METHOD PUBLIC Check_LWORD_TO_BOOL_Max
VAR
	value : LWORD := DatatypeLimits.LWORD_MAX_VALUE;
	actual : BOOL;
	converted : BOOL;
	equal : BOOL;
END_VAR
TEST('Check_LWORD_TO_BOOL_Max');

// @TEST-RUN
converted := TryConvert_LWORD_TO_Destination(value, actual);
equal := actual = LWORD_TO_BOOL(value);

// @TEST-ASSERT
AssertTrue(Condition := equal, Message := 'Did not convert LWORD to BOOL correctly');
AssertTrue(Condition := converted, Message := 'Did not report LWORD to BOOL conversion was successful');

TEST_FINISHED();
END_METHOD

METHOD PUBLIC Check_LWORD_TO_BYTE_Min
VAR
	value : LWORD := DatatypeLimits.LWORD_MIN_VALUE;
	actual : BYTE;
	converted : BOOL;
	equal : BOOL;
END_VAR
TEST('Check_LWORD_TO_BYTE_Min');

// @TEST-RUN
converted := TryConvert_LWORD_TO_Destination(value, actual);
equal := actual = LWORD_TO_BYTE(value);

// @TEST-ASSERT
AssertTrue(Condition := equal, Message := 'Did not convert LWORD to BYTE correctly');
AssertTrue(Condition := converted, Message := 'Did not report LWORD to BYTE conversion was successful');

TEST_FINISHED();
END_METHOD

METHOD PUBLIC Check_LWORD_TO_BYTE_TooHigh
VAR
	value : LWORD := DatatypeLimits.LWORD_MAX_VALUE;
	actual : BYTE;
	converted : BOOL;
END_VAR
TEST('Check_LWORD_TO_BYTE_TooHigh');

// @TEST-RUN
converted := TryConvert_LWORD_TO_Destination(value, actual);

// @TEST-ASSERT
AssertFalse(Condition := converted, Message := 'Did not report LWORD to BYTE conversion was prevented');

TEST_FINISHED();
END_METHOD

METHOD PUBLIC Check_LWORD_TO_BYTE_Max
VAR
	value : LWORD := DatatypeLimits.MAX_VALUE_OF_LWORD_WHICH_CAN_BE_HELD_IN_A_BYTE;
	actual : BYTE;
	converted : BOOL;
	equal : BOOL;
END_VAR
TEST('Check_LWORD_TO_BYTE_Max');

// @TEST-RUN
converted := TryConvert_LWORD_TO_Destination(value, actual);
equal := actual = LWORD_TO_BYTE(value);

// @TEST-ASSERT
AssertTrue(Condition := equal, Message := 'Did not convert LWORD to BYTE correctly');
AssertTrue(Condition := converted, Message := 'Did not report LWORD to BYTE conversion was successful');

TEST_FINISHED();
END_METHOD

METHOD PUBLIC Check_LWORD_TO_DATE_Min
VAR
	value : LWORD := DatatypeLimits.LWORD_MIN_VALUE;
	actual : DATE;
	converted : BOOL;
	equal : BOOL;
END_VAR
TEST('Check_LWORD_TO_DATE_Min');

// @TEST-RUN
converted := TryConvert_LWORD_TO_Destination(value, actual);
equal := actual = LWORD_TO_DATE(value);

// @TEST-ASSERT
AssertTrue(Condition := equal, Message := 'Did not convert LWORD to DATE correctly');
AssertTrue(Condition := converted, Message := 'Did not report LWORD to DATE conversion was successful');

TEST_FINISHED();
END_METHOD

METHOD PUBLIC Check_LWORD_TO_DATE_TooHigh
VAR
	value : LWORD := DatatypeLimits.LWORD_MAX_VALUE;
	actual : DATE;
	converted : BOOL;
END_VAR
TEST('Check_LWORD_TO_DATE_TooHigh');

// @TEST-RUN
converted := TryConvert_LWORD_TO_Destination(value, actual);

// @TEST-ASSERT
AssertFalse(Condition := converted, Message := 'Did not report LWORD to DATE conversion was prevented');

TEST_FINISHED();
END_METHOD

METHOD PUBLIC Check_LWORD_TO_DATE_Max
VAR
	value : LWORD := DatatypeLimits.MAX_VALUE_OF_LWORD_WHICH_CAN_BE_HELD_IN_A_DATE;
	actual : DATE;
	converted : BOOL;
	equal : BOOL;
END_VAR
TEST('Check_LWORD_TO_DATE_Max');

// @TEST-RUN
converted := TryConvert_LWORD_TO_Destination(value, actual);
equal := actual = LWORD_TO_DATE(value);

// @TEST-ASSERT
AssertTrue(Condition := equal, Message := 'Did not convert LWORD to DATE correctly');
AssertTrue(Condition := converted, Message := 'Did not report LWORD to DATE conversion was successful');

TEST_FINISHED();
END_METHOD

METHOD PUBLIC Check_LWORD_TO_DINT_Min
VAR
	value : LWORD := DatatypeLimits.LWORD_MIN_VALUE;
	actual : DINT;
	converted : BOOL;
	equal : BOOL;
END_VAR
TEST('Check_LWORD_TO_DINT_Min');

// @TEST-RUN
converted := TryConvert_LWORD_TO_Destination(value, actual);
equal := actual = LWORD_TO_DINT(value);

// @TEST-ASSERT
AssertTrue(Condition := equal, Message := 'Did not convert LWORD to DINT correctly');
AssertTrue(Condition := converted, Message := 'Did not report LWORD to DINT conversion was successful');

TEST_FINISHED();
END_METHOD

METHOD PUBLIC Check_LWORD_TO_DINT_TooHigh
VAR
	value : LWORD := DatatypeLimits.LWORD_MAX_VALUE;
	actual : DINT;
	converted : BOOL;
END_VAR
TEST('Check_LWORD_TO_DINT_TooHigh');

// @TEST-RUN
converted := TryConvert_LWORD_TO_Destination(value, actual);

// @TEST-ASSERT
AssertFalse(Condition := converted, Message := 'Did not report LWORD to DINT conversion was prevented');

TEST_FINISHED();
END_METHOD

METHOD PUBLIC Check_LWORD_TO_DINT_Max
VAR
	value : LWORD := DatatypeLimits.MAX_VALUE_OF_LWORD_WHICH_CAN_BE_HELD_IN_A_DINT;
	actual : DINT;
	converted : BOOL;
	equal : BOOL;
END_VAR
TEST('Check_LWORD_TO_DINT_Max');

// @TEST-RUN
converted := TryConvert_LWORD_TO_Destination(value, actual);
equal := actual = LWORD_TO_DINT(value);

// @TEST-ASSERT
AssertTrue(Condition := equal, Message := 'Did not convert LWORD to DINT correctly');
AssertTrue(Condition := converted, Message := 'Did not report LWORD to DINT conversion was successful');

TEST_FINISHED();
END_METHOD

METHOD PUBLIC Check_LWORD_TO_DT_Min
VAR
	value : LWORD := DatatypeLimits.LWORD_MIN_VALUE;
	actual : DT;
	converted : BOOL;
	equal : BOOL;
END_VAR
TEST('Check_LWORD_TO_DT_Min');

// @TEST-RUN
converted := TryConvert_LWORD_TO_Destination(value, actual);
equal := actual = LWORD_TO_DT(value);

// @TEST-ASSERT
AssertTrue(Condition := equal, Message := 'Did not convert LWORD to DT correctly');
AssertTrue(Condition := converted, Message := 'Did not report LWORD to DT conversion was successful');

TEST_FINISHED();
END_METHOD

METHOD PUBLIC Check_LWORD_TO_DT_TooHigh
VAR
	value : LWORD := DatatypeLimits.LWORD_MAX_VALUE;
	actual : DT;
	converted : BOOL;
END_VAR
TEST('Check_LWORD_TO_DT_TooHigh');

// @TEST-RUN
converted := TryConvert_LWORD_TO_Destination(value, actual);

// @TEST-ASSERT
AssertFalse(Condition := converted, Message := 'Did not report LWORD to DT conversion was prevented');

TEST_FINISHED();
END_METHOD

METHOD PUBLIC Check_LWORD_TO_DT_Max
VAR
	value : LWORD := DatatypeLimits.MAX_VALUE_OF_LWORD_WHICH_CAN_BE_HELD_IN_A_DT;
	actual : DT;
	converted : BOOL;
	equal : BOOL;
END_VAR
TEST('Check_LWORD_TO_DT_Max');

// @TEST-RUN
converted := TryConvert_LWORD_TO_Destination(value, actual);
equal := actual = LWORD_TO_DT(value);

// @TEST-ASSERT
AssertTrue(Condition := equal, Message := 'Did not convert LWORD to DT correctly');
AssertTrue(Condition := converted, Message := 'Did not report LWORD to DT conversion was successful');

TEST_FINISHED();
END_METHOD

METHOD PUBLIC Check_LWORD_TO_DWORD_Min
VAR
	value : LWORD := DatatypeLimits.LWORD_MIN_VALUE;
	actual : DWORD;
	converted : BOOL;
	equal : BOOL;
END_VAR
TEST('Check_LWORD_TO_DWORD_Min');

// @TEST-RUN
converted := TryConvert_LWORD_TO_Destination(value, actual);
equal := actual = LWORD_TO_DWORD(value);

// @TEST-ASSERT
AssertTrue(Condition := equal, Message := 'Did not convert LWORD to DWORD correctly');
AssertTrue(Condition := converted, Message := 'Did not report LWORD to DWORD conversion was successful');

TEST_FINISHED();
END_METHOD

METHOD PUBLIC Check_LWORD_TO_DWORD_TooHigh
VAR
	value : LWORD := DatatypeLimits.LWORD_MAX_VALUE;
	actual : DWORD;
	converted : BOOL;
END_VAR
TEST('Check_LWORD_TO_DWORD_TooHigh');

// @TEST-RUN
converted := TryConvert_LWORD_TO_Destination(value, actual);

// @TEST-ASSERT
AssertFalse(Condition := converted, Message := 'Did not report LWORD to DWORD conversion was prevented');

TEST_FINISHED();
END_METHOD

METHOD PUBLIC Check_LWORD_TO_DWORD_Max
VAR
	value : LWORD := DatatypeLimits.MAX_VALUE_OF_LWORD_WHICH_CAN_BE_HELD_IN_A_DWORD;
	actual : DWORD;
	converted : BOOL;
	equal : BOOL;
END_VAR
TEST('Check_LWORD_TO_DWORD_Max');

// @TEST-RUN
converted := TryConvert_LWORD_TO_Destination(value, actual);
equal := actual = LWORD_TO_DWORD(value);

// @TEST-ASSERT
AssertTrue(Condition := equal, Message := 'Did not convert LWORD to DWORD correctly');
AssertTrue(Condition := converted, Message := 'Did not report LWORD to DWORD conversion was successful');

TEST_FINISHED();
END_METHOD

METHOD PUBLIC Check_LWORD_TO_INT_Min
VAR
	value : LWORD := DatatypeLimits.LWORD_MIN_VALUE;
	actual : INT;
	converted : BOOL;
	equal : BOOL;
END_VAR
TEST('Check_LWORD_TO_INT_Min');

// @TEST-RUN
converted := TryConvert_LWORD_TO_Destination(value, actual);
equal := actual = LWORD_TO_INT(value);

// @TEST-ASSERT
AssertTrue(Condition := equal, Message := 'Did not convert LWORD to INT correctly');
AssertTrue(Condition := converted, Message := 'Did not report LWORD to INT conversion was successful');

TEST_FINISHED();
END_METHOD

METHOD PUBLIC Check_LWORD_TO_INT_TooHigh
VAR
	value : LWORD := DatatypeLimits.LWORD_MAX_VALUE;
	actual : INT;
	converted : BOOL;
END_VAR
TEST('Check_LWORD_TO_INT_TooHigh');

// @TEST-RUN
converted := TryConvert_LWORD_TO_Destination(value, actual);

// @TEST-ASSERT
AssertFalse(Condition := converted, Message := 'Did not report LWORD to INT conversion was prevented');

TEST_FINISHED();
END_METHOD

METHOD PUBLIC Check_LWORD_TO_INT_Max
VAR
	value : LWORD := DatatypeLimits.MAX_VALUE_OF_LWORD_WHICH_CAN_BE_HELD_IN_A_INT;
	actual : INT;
	converted : BOOL;
	equal : BOOL;
END_VAR
TEST('Check_LWORD_TO_INT_Max');

// @TEST-RUN
converted := TryConvert_LWORD_TO_Destination(value, actual);
equal := actual = LWORD_TO_INT(value);

// @TEST-ASSERT
AssertTrue(Condition := equal, Message := 'Did not convert LWORD to INT correctly');
AssertTrue(Condition := converted, Message := 'Did not report LWORD to INT conversion was successful');

TEST_FINISHED();
END_METHOD

METHOD PUBLIC Check_LWORD_TO_LINT_Min
VAR
	value : LWORD := DatatypeLimits.LWORD_MIN_VALUE;
	actual : LINT;
	converted : BOOL;
	equal : BOOL;
END_VAR
TEST('Check_LWORD_TO_LINT_Min');

// @TEST-RUN
converted := TryConvert_LWORD_TO_Destination(value, actual);
equal := actual = LWORD_TO_LINT(value);

// @TEST-ASSERT
AssertTrue(Condition := equal, Message := 'Did not convert LWORD to LINT correctly');
AssertTrue(Condition := converted, Message := 'Did not report LWORD to LINT conversion was successful');

TEST_FINISHED();
END_METHOD

METHOD PUBLIC Check_LWORD_TO_LINT_TooHigh
VAR
	value : LWORD := DatatypeLimits.LWORD_MAX_VALUE;
	actual : LINT;
	converted : BOOL;
END_VAR
TEST('Check_LWORD_TO_LINT_TooHigh');

// @TEST-RUN
converted := TryConvert_LWORD_TO_Destination(value, actual);

// @TEST-ASSERT
AssertFalse(Condition := converted, Message := 'Did not report LWORD to LINT conversion was prevented');

TEST_FINISHED();
END_METHOD

METHOD PUBLIC Check_LWORD_TO_LINT_Max
VAR
	value : LWORD := DatatypeLimits.MAX_VALUE_OF_LWORD_WHICH_CAN_BE_HELD_IN_A_LINT;
	actual : LINT;
	converted : BOOL;
	equal : BOOL;
END_VAR
TEST('Check_LWORD_TO_LINT_Max');

// @TEST-RUN
converted := TryConvert_LWORD_TO_Destination(value, actual);
equal := actual = LWORD_TO_LINT(value);

// @TEST-ASSERT
AssertTrue(Condition := equal, Message := 'Did not convert LWORD to LINT correctly');
AssertTrue(Condition := converted, Message := 'Did not report LWORD to LINT conversion was successful');

TEST_FINISHED();
END_METHOD

METHOD PUBLIC Check_LWORD_TO_LREAL_Min
VAR
	value : LWORD := DatatypeLimits.LWORD_MIN_VALUE;
	actual : LREAL;
	converted : BOOL;
	equal : BOOL;
END_VAR
TEST('Check_LWORD_TO_LREAL_Min');

// @TEST-RUN
converted := TryConvert_LWORD_TO_Destination(value, actual);
equal := actual = LWORD_TO_LREAL(value);

// @TEST-ASSERT
AssertTrue(Condition := equal, Message := 'Did not convert LWORD to LREAL correctly');
AssertTrue(Condition := converted, Message := 'Did not report LWORD to LREAL conversion was successful');

TEST_FINISHED();
END_METHOD

METHOD PUBLIC Check_LWORD_TO_LREAL_Max
VAR
	value : LWORD := DatatypeLimits.LWORD_MAX_VALUE;
	actual : LREAL;
	converted : BOOL;
	equal : BOOL;
END_VAR
TEST('Check_LWORD_TO_LREAL_Max');

// @TEST-RUN
converted := TryConvert_LWORD_TO_Destination(value, actual);
equal := actual = LWORD_TO_LREAL(value);

// @TEST-ASSERT
AssertTrue(Condition := equal, Message := 'Did not convert LWORD to LREAL correctly');
AssertTrue(Condition := converted, Message := 'Did not report LWORD to LREAL conversion was successful');

TEST_FINISHED();
END_METHOD

METHOD PUBLIC Check_LWORD_TO_LWORD_Min
VAR
	value : LWORD := DatatypeLimits.LWORD_MIN_VALUE;
	actual : LWORD;
	converted : BOOL;
	equal : BOOL;
END_VAR
TEST('Check_LWORD_TO_LWORD_Min');

// @TEST-RUN
converted := TryConvert_LWORD_TO_Destination(value, actual);
equal := actual = value;

// @TEST-ASSERT
AssertTrue(Condition := equal, Message := 'Did not convert LWORD to LWORD correctly');
AssertTrue(Condition := converted, Message := 'Did not report LWORD to LWORD conversion was successful');

TEST_FINISHED();
END_METHOD

METHOD PUBLIC Check_LWORD_TO_LWORD_Max
VAR
	value : LWORD := DatatypeLimits.LWORD_MAX_VALUE;
	actual : LWORD;
	converted : BOOL;
	equal : BOOL;
END_VAR
TEST('Check_LWORD_TO_LWORD_Max');

// @TEST-RUN
converted := TryConvert_LWORD_TO_Destination(value, actual);
equal := actual = value;

// @TEST-ASSERT
AssertTrue(Condition := equal, Message := 'Did not convert LWORD to LWORD correctly');
AssertTrue(Condition := converted, Message := 'Did not report LWORD to LWORD conversion was successful');

TEST_FINISHED();
END_METHOD

METHOD PUBLIC Check_LWORD_TO_REAL_Min
VAR
	value : LWORD := DatatypeLimits.LWORD_MIN_VALUE;
	actual : REAL;
	converted : BOOL;
	equal : BOOL;
END_VAR
TEST('Check_LWORD_TO_REAL_Min');

// @TEST-RUN
converted := TryConvert_LWORD_TO_Destination(value, actual);
equal := actual = LWORD_TO_REAL(value);

// @TEST-ASSERT
AssertTrue(Condition := equal, Message := 'Did not convert LWORD to REAL correctly');
AssertTrue(Condition := converted, Message := 'Did not report LWORD to REAL conversion was successful');

TEST_FINISHED();
END_METHOD

METHOD PUBLIC Check_LWORD_TO_REAL_Max
VAR
	value : LWORD := DatatypeLimits.LWORD_MAX_VALUE;
	actual : REAL;
	converted : BOOL;
	equal : BOOL;
END_VAR
TEST('Check_LWORD_TO_REAL_Max');

// @TEST-RUN
converted := TryConvert_LWORD_TO_Destination(value, actual);
equal := actual = LWORD_TO_REAL(value);

// @TEST-ASSERT
AssertTrue(Condition := equal, Message := 'Did not convert LWORD to REAL correctly');
AssertTrue(Condition := converted, Message := 'Did not report LWORD to REAL conversion was successful');

TEST_FINISHED();
END_METHOD

METHOD PUBLIC Check_LWORD_TO_SINT_Min
VAR
	value : LWORD := DatatypeLimits.LWORD_MIN_VALUE;
	actual : SINT;
	converted : BOOL;
	equal : BOOL;
END_VAR
TEST('Check_LWORD_TO_SINT_Min');

// @TEST-RUN
converted := TryConvert_LWORD_TO_Destination(value, actual);
equal := actual = LWORD_TO_SINT(value);

// @TEST-ASSERT
AssertTrue(Condition := equal, Message := 'Did not convert LWORD to SINT correctly');
AssertTrue(Condition := converted, Message := 'Did not report LWORD to SINT conversion was successful');

TEST_FINISHED();
END_METHOD

METHOD PUBLIC Check_LWORD_TO_SINT_TooHigh
VAR
	value : LWORD := DatatypeLimits.LWORD_MAX_VALUE;
	actual : SINT;
	converted : BOOL;
END_VAR
TEST('Check_LWORD_TO_SINT_TooHigh');

// @TEST-RUN
converted := TryConvert_LWORD_TO_Destination(value, actual);

// @TEST-ASSERT
AssertFalse(Condition := converted, Message := 'Did not report LWORD to SINT conversion was prevented');

TEST_FINISHED();
END_METHOD

METHOD PUBLIC Check_LWORD_TO_SINT_Max
VAR
	value : LWORD := DatatypeLimits.MAX_VALUE_OF_LWORD_WHICH_CAN_BE_HELD_IN_A_SINT;
	actual : SINT;
	converted : BOOL;
	equal : BOOL;
END_VAR
TEST('Check_LWORD_TO_SINT_Max');

// @TEST-RUN
converted := TryConvert_LWORD_TO_Destination(value, actual);
equal := actual = LWORD_TO_SINT(value);

// @TEST-ASSERT
AssertTrue(Condition := equal, Message := 'Did not convert LWORD to SINT correctly');
AssertTrue(Condition := converted, Message := 'Did not report LWORD to SINT conversion was successful');

TEST_FINISHED();
END_METHOD

METHOD PUBLIC Check_LWORD_TO_STRING_Min
VAR
	value : LWORD := DatatypeLimits.LWORD_MIN_VALUE;
	actual : STRING;
	converted : BOOL;
	equal : BOOL;
END_VAR
TEST('Check_LWORD_TO_STRING_Min');

// @TEST-RUN
converted := TryConvert_LWORD_TO_Destination(value, actual);
equal := actual = LWORD_TO_STRING(value);

// @TEST-ASSERT
AssertTrue(Condition := equal, Message := 'Did not convert LWORD to STRING correctly');
AssertTrue(Condition := converted, Message := 'Did not report LWORD to STRING conversion was successful');

TEST_FINISHED();
END_METHOD

METHOD PUBLIC Check_LWORD_TO_STRING_Max
VAR
	value : LWORD := DatatypeLimits.LWORD_MAX_VALUE;
	actual : STRING;
	converted : BOOL;
	equal : BOOL;
END_VAR
TEST('Check_LWORD_TO_STRING_Max');

// @TEST-RUN
converted := TryConvert_LWORD_TO_Destination(value, actual);
equal := actual = LWORD_TO_STRING(value);

// @TEST-ASSERT
AssertTrue(Condition := equal, Message := 'Did not convert LWORD to STRING correctly');
AssertTrue(Condition := converted, Message := 'Did not report LWORD to STRING conversion was successful');

TEST_FINISHED();
END_METHOD

METHOD PUBLIC Check_LWORD_TO_TIME_Min
VAR
	value : LWORD := DatatypeLimits.LWORD_MIN_VALUE;
	actual : TIME;
	converted : BOOL;
	equal : BOOL;
END_VAR
TEST('Check_LWORD_TO_TIME_Min');

// @TEST-RUN
converted := TryConvert_LWORD_TO_Destination(value, actual);
equal := actual = LWORD_TO_TIME(value);

// @TEST-ASSERT
AssertTrue(Condition := equal, Message := 'Did not convert LWORD to TIME correctly');
AssertTrue(Condition := converted, Message := 'Did not report LWORD to TIME conversion was successful');

TEST_FINISHED();
END_METHOD

METHOD PUBLIC Check_LWORD_TO_TIME_TooHigh
VAR
	value : LWORD := DatatypeLimits.LWORD_MAX_VALUE;
	actual : TIME;
	converted : BOOL;
END_VAR
TEST('Check_LWORD_TO_TIME_TooHigh');

// @TEST-RUN
converted := TryConvert_LWORD_TO_Destination(value, actual);

// @TEST-ASSERT
AssertFalse(Condition := converted, Message := 'Did not report LWORD to TIME conversion was prevented');

TEST_FINISHED();
END_METHOD

METHOD PUBLIC Check_LWORD_TO_TIME_Max
VAR
	value : LWORD := DatatypeLimits.MAX_VALUE_OF_LWORD_WHICH_CAN_BE_HELD_IN_A_TIME;
	actual : TIME;
	converted : BOOL;
	equal : BOOL;
END_VAR
TEST('Check_LWORD_TO_TIME_Max');

// @TEST-RUN
converted := TryConvert_LWORD_TO_Destination(value, actual);
equal := actual = LWORD_TO_TIME(value);

// @TEST-ASSERT
AssertTrue(Condition := equal, Message := 'Did not convert LWORD to TIME correctly');
AssertTrue(Condition := converted, Message := 'Did not report LWORD to TIME conversion was successful');

TEST_FINISHED();
END_METHOD

METHOD PUBLIC Check_LWORD_TO_TOD_Min
VAR
	value : LWORD := DatatypeLimits.LWORD_MIN_VALUE;
	actual : TOD;
	converted : BOOL;
	equal : BOOL;
END_VAR
TEST('Check_LWORD_TO_TOD_Min');

// @TEST-RUN
converted := TryConvert_LWORD_TO_Destination(value, actual);
equal := actual = LWORD_TO_TOD(value);

// @TEST-ASSERT
AssertTrue(Condition := equal, Message := 'Did not convert LWORD to TOD correctly');
AssertTrue(Condition := converted, Message := 'Did not report LWORD to TOD conversion was successful');

TEST_FINISHED();
END_METHOD

METHOD PUBLIC Check_LWORD_TO_TOD_TooHigh
VAR
	value : LWORD := DatatypeLimits.LWORD_MAX_VALUE;
	actual : TOD;
	converted : BOOL;
END_VAR
TEST('Check_LWORD_TO_TOD_TooHigh');

// @TEST-RUN
converted := TryConvert_LWORD_TO_Destination(value, actual);

// @TEST-ASSERT
AssertFalse(Condition := converted, Message := 'Did not report LWORD to TOD conversion was prevented');

TEST_FINISHED();
END_METHOD

METHOD PUBLIC Check_LWORD_TO_TOD_Max
VAR
	value : LWORD := DatatypeLimits.MAX_VALUE_OF_LWORD_WHICH_CAN_BE_HELD_IN_A_TOD;
	actual : TOD;
	converted : BOOL;
	equal : BOOL;
END_VAR
TEST('Check_LWORD_TO_TOD_Max');

// @TEST-RUN
converted := TryConvert_LWORD_TO_Destination(value, actual);
equal := actual = LWORD_TO_TOD(value);

// @TEST-ASSERT
AssertTrue(Condition := equal, Message := 'Did not convert LWORD to TOD correctly');
AssertTrue(Condition := converted, Message := 'Did not report LWORD to TOD conversion was successful');

TEST_FINISHED();
END_METHOD

METHOD PUBLIC Check_LWORD_TO_UDINT_Min
VAR
	value : LWORD := DatatypeLimits.LWORD_MIN_VALUE;
	actual : UDINT;
	converted : BOOL;
	equal : BOOL;
END_VAR
TEST('Check_LWORD_TO_UDINT_Min');

// @TEST-RUN
converted := TryConvert_LWORD_TO_Destination(value, actual);
equal := actual = LWORD_TO_UDINT(value);

// @TEST-ASSERT
AssertTrue(Condition := equal, Message := 'Did not convert LWORD to UDINT correctly');
AssertTrue(Condition := converted, Message := 'Did not report LWORD to UDINT conversion was successful');

TEST_FINISHED();
END_METHOD

METHOD PUBLIC Check_LWORD_TO_UDINT_TooHigh
VAR
	value : LWORD := DatatypeLimits.LWORD_MAX_VALUE;
	actual : UDINT;
	converted : BOOL;
END_VAR
TEST('Check_LWORD_TO_UDINT_TooHigh');

// @TEST-RUN
converted := TryConvert_LWORD_TO_Destination(value, actual);

// @TEST-ASSERT
AssertFalse(Condition := converted, Message := 'Did not report LWORD to UDINT conversion was prevented');

TEST_FINISHED();
END_METHOD

METHOD PUBLIC Check_LWORD_TO_UDINT_Max
VAR
	value : LWORD := DatatypeLimits.MAX_VALUE_OF_LWORD_WHICH_CAN_BE_HELD_IN_A_UDINT;
	actual : UDINT;
	converted : BOOL;
	equal : BOOL;
END_VAR
TEST('Check_LWORD_TO_UDINT_Max');

// @TEST-RUN
converted := TryConvert_LWORD_TO_Destination(value, actual);
equal := actual = LWORD_TO_UDINT(value);

// @TEST-ASSERT
AssertTrue(Condition := equal, Message := 'Did not convert LWORD to UDINT correctly');
AssertTrue(Condition := converted, Message := 'Did not report LWORD to UDINT conversion was successful');

TEST_FINISHED();
END_METHOD

METHOD PUBLIC Check_LWORD_TO_UINT_Min
VAR
	value : LWORD := DatatypeLimits.LWORD_MIN_VALUE;
	actual : UINT;
	converted : BOOL;
	equal : BOOL;
END_VAR
TEST('Check_LWORD_TO_UINT_Min');

// @TEST-RUN
converted := TryConvert_LWORD_TO_Destination(value, actual);
equal := actual = LWORD_TO_UINT(value);

// @TEST-ASSERT
AssertTrue(Condition := equal, Message := 'Did not convert LWORD to UINT correctly');
AssertTrue(Condition := converted, Message := 'Did not report LWORD to UINT conversion was successful');

TEST_FINISHED();
END_METHOD

METHOD PUBLIC Check_LWORD_TO_UINT_TooHigh
VAR
	value : LWORD := DatatypeLimits.LWORD_MAX_VALUE;
	actual : UINT;
	converted : BOOL;
END_VAR
TEST('Check_LWORD_TO_UINT_TooHigh');

// @TEST-RUN
converted := TryConvert_LWORD_TO_Destination(value, actual);

// @TEST-ASSERT
AssertFalse(Condition := converted, Message := 'Did not report LWORD to UINT conversion was prevented');

TEST_FINISHED();
END_METHOD

METHOD PUBLIC Check_LWORD_TO_UINT_Max
VAR
	value : LWORD := DatatypeLimits.MAX_VALUE_OF_LWORD_WHICH_CAN_BE_HELD_IN_A_UINT;
	actual : UINT;
	converted : BOOL;
	equal : BOOL;
END_VAR
TEST('Check_LWORD_TO_UINT_Max');

// @TEST-RUN
converted := TryConvert_LWORD_TO_Destination(value, actual);
equal := actual = LWORD_TO_UINT(value);

// @TEST-ASSERT
AssertTrue(Condition := equal, Message := 'Did not convert LWORD to UINT correctly');
AssertTrue(Condition := converted, Message := 'Did not report LWORD to UINT conversion was successful');

TEST_FINISHED();
END_METHOD

METHOD PUBLIC Check_LWORD_TO_ULINT_Min
VAR
	value : LWORD := DatatypeLimits.LWORD_MIN_VALUE;
	actual : ULINT;
	converted : BOOL;
	equal : BOOL;
END_VAR
TEST('Check_LWORD_TO_ULINT_Min');

// @TEST-RUN
converted := TryConvert_LWORD_TO_Destination(value, actual);
equal := actual = LWORD_TO_ULINT(value);

// @TEST-ASSERT
AssertTrue(Condition := equal, Message := 'Did not convert LWORD to ULINT correctly');
AssertTrue(Condition := converted, Message := 'Did not report LWORD to ULINT conversion was successful');

TEST_FINISHED();
END_METHOD

METHOD PUBLIC Check_LWORD_TO_ULINT_Max
VAR
	value : LWORD := DatatypeLimits.LWORD_MAX_VALUE;
	actual : ULINT;
	converted : BOOL;
	equal : BOOL;
END_VAR
TEST('Check_LWORD_TO_ULINT_Max');

// @TEST-RUN
converted := TryConvert_LWORD_TO_Destination(value, actual);
equal := actual = LWORD_TO_ULINT(value);

// @TEST-ASSERT
AssertTrue(Condition := equal, Message := 'Did not convert LWORD to ULINT correctly');
AssertTrue(Condition := converted, Message := 'Did not report LWORD to ULINT conversion was successful');

TEST_FINISHED();
END_METHOD

METHOD PUBLIC Check_LWORD_TO_USINT_Min
VAR
	value : LWORD := DatatypeLimits.LWORD_MIN_VALUE;
	actual : USINT;
	converted : BOOL;
	equal : BOOL;
END_VAR
TEST('Check_LWORD_TO_USINT_Min');

// @TEST-RUN
converted := TryConvert_LWORD_TO_Destination(value, actual);
equal := actual = LWORD_TO_USINT(value);

// @TEST-ASSERT
AssertTrue(Condition := equal, Message := 'Did not convert LWORD to USINT correctly');
AssertTrue(Condition := converted, Message := 'Did not report LWORD to USINT conversion was successful');

TEST_FINISHED();
END_METHOD

METHOD PUBLIC Check_LWORD_TO_USINT_TooHigh
VAR
	value : LWORD := DatatypeLimits.LWORD_MAX_VALUE;
	actual : USINT;
	converted : BOOL;
END_VAR
TEST('Check_LWORD_TO_USINT_TooHigh');

// @TEST-RUN
converted := TryConvert_LWORD_TO_Destination(value, actual);

// @TEST-ASSERT
AssertFalse(Condition := converted, Message := 'Did not report LWORD to USINT conversion was prevented');

TEST_FINISHED();
END_METHOD

METHOD PUBLIC Check_LWORD_TO_USINT_Max
VAR
	value : LWORD := DatatypeLimits.MAX_VALUE_OF_LWORD_WHICH_CAN_BE_HELD_IN_A_USINT;
	actual : USINT;
	converted : BOOL;
	equal : BOOL;
END_VAR
TEST('Check_LWORD_TO_USINT_Max');

// @TEST-RUN
converted := TryConvert_LWORD_TO_Destination(value, actual);
equal := actual = LWORD_TO_USINT(value);

// @TEST-ASSERT
AssertTrue(Condition := equal, Message := 'Did not convert LWORD to USINT correctly');
AssertTrue(Condition := converted, Message := 'Did not report LWORD to USINT conversion was successful');

TEST_FINISHED();
END_METHOD

METHOD PUBLIC Check_LWORD_TO_WORD_Min
VAR
	value : LWORD := DatatypeLimits.LWORD_MIN_VALUE;
	actual : WORD;
	converted : BOOL;
	equal : BOOL;
END_VAR
TEST('Check_LWORD_TO_WORD_Min');

// @TEST-RUN
converted := TryConvert_LWORD_TO_Destination(value, actual);
equal := actual = LWORD_TO_WORD(value);

// @TEST-ASSERT
AssertTrue(Condition := equal, Message := 'Did not convert LWORD to WORD correctly');
AssertTrue(Condition := converted, Message := 'Did not report LWORD to WORD conversion was successful');

TEST_FINISHED();
END_METHOD

METHOD PUBLIC Check_LWORD_TO_WORD_TooHigh
VAR
	value : LWORD := DatatypeLimits.LWORD_MAX_VALUE;
	actual : WORD;
	converted : BOOL;
END_VAR
TEST('Check_LWORD_TO_WORD_TooHigh');

// @TEST-RUN
converted := TryConvert_LWORD_TO_Destination(value, actual);

// @TEST-ASSERT
AssertFalse(Condition := converted, Message := 'Did not report LWORD to WORD conversion was prevented');

TEST_FINISHED();
END_METHOD

METHOD PUBLIC Check_LWORD_TO_WORD_Max
VAR
	value : LWORD := DatatypeLimits.MAX_VALUE_OF_LWORD_WHICH_CAN_BE_HELD_IN_A_WORD;
	actual : WORD;
	converted : BOOL;
	equal : BOOL;
END_VAR
TEST('Check_LWORD_TO_WORD_Max');

// @TEST-RUN
converted := TryConvert_LWORD_TO_Destination(value, actual);
equal := actual = LWORD_TO_WORD(value);

// @TEST-ASSERT
AssertTrue(Condition := equal, Message := 'Did not convert LWORD to WORD correctly');
AssertTrue(Condition := converted, Message := 'Did not report LWORD to WORD conversion was successful');

TEST_FINISHED();
END_METHOD

END_FUNCTION_BLOCK

// ---- Tests/SINT_TO_TestSuite.TcPOU
FUNCTION_BLOCK PUBLIC SINT_TO_TestSuite EXTENDS TcUnit.FB_TestSuite
VAR
END_VAR

Check_SINT_TO_BOOL_Max();
Check_SINT_TO_BOOL_Min();
Check_SINT_TO_BYTE_Max();
Check_SINT_TO_BYTE_Min();
Check_SINT_TO_BYTE_TooLow();
Check_SINT_TO_WORD_Max();
Check_SINT_TO_WORD_Min();
Check_SINT_TO_WORD_TooLow();
Check_SINT_TO_DWORD_Max();
Check_SINT_TO_DWORD_Min();
Check_SINT_TO_DWORD_TooLow();
Check_SINT_TO_LWORD_Max();
Check_SINT_TO_LWORD_Min();
Check_SINT_TO_LWORD_TooLow();
Check_SINT_TO_SINT_Max();
Check_SINT_TO_SINT_Min();
Check_SINT_TO_INT_Max();
Check_SINT_TO_INT_Min();
Check_SINT_TO_DINT_Max();
Check_SINT_TO_DINT_Min();
Check_SINT_TO_LINT_Max();
Check_SINT_TO_LINT_Min();
Check_SINT_TO_USINT_Max();
Check_SINT_TO_USINT_Min();
Check_SINT_TO_USINT_TooLow();
Check_SINT_TO_UINT_Max();
Check_SINT_TO_UINT_Min();
Check_SINT_TO_UINT_TooLow();
Check_SINT_TO_UDINT_Max();
Check_SINT_TO_UDINT_Min();
Check_SINT_TO_UDINT_TooLow();
Check_SINT_TO_ULINT_Max();
Check_SINT_TO_ULINT_Min();
Check_SINT_TO_ULINT_TooLow();
Check_SINT_TO_REAL_Max();
Check_SINT_TO_REAL_Min();
Check_SINT_TO_LREAL_Max();
Check_SINT_TO_LREAL_Min();
Check_SINT_TO_TIME_Max();
Check_SINT_TO_TIME_Min();
Check_SINT_TO_TIME_TooLow();
Check_SINT_TO_TOD_Max();
Check_SINT_TO_TOD_Min();
Check_SINT_TO_TOD_TooLow();
Check_SINT_TO_DATE_Max();
Check_SINT_TO_DATE_Min();
Check_SINT_TO_DATE_TooLow();
Check_SINT_TO_DT_Max();
Check_SINT_TO_DT_Min();
Check_SINT_TO_DT_TooLow();
Check_SINT_TO_STRING_Max();
Check_SINT_TO_STRING_Min();

METHOD PUBLIC Check_SINT_TO_BOOL_Min
VAR
	value : SINT := DatatypeLimits.SINT_MIN_VALUE;
	actual : BOOL;
	converted : BOOL;
	equal : BOOL;
END_VAR
TEST('Check_SINT_TO_BOOL_Min');

// @TEST-RUN
converted := TryConvert_SINT_TO_Destination(value, actual);
equal := actual = SINT_TO_BOOL(value);

// @TEST-ASSERT
AssertTrue(Condition := equal, Message := 'Did not convert SINT to BOOL correctly');
AssertTrue(Condition := converted, Message := 'Did not report SINT to BOOL conversion was successful');

TEST_FINISHED();
END_METHOD

METHOD PUBLIC Check_SINT_TO_BOOL_Max
VAR
	value : SINT := DatatypeLimits.SINT_MAX_VALUE;
	actual : BOOL;
	converted : BOOL;
	equal : BOOL;
END_VAR
TEST('Check_SINT_TO_BOOL_Max');

// @TEST-RUN
converted := TryConvert_SINT_TO_Destination(value, actual);
equal := actual = SINT_TO_BOOL(value);

// @TEST-ASSERT
AssertTrue(Condition := equal, Message := 'Did not convert SINT to BOOL correctly');
AssertTrue(Condition := converted, Message := 'Did not report SINT to BOOL conversion was successful');

TEST_FINISHED();
END_METHOD

METHOD PUBLIC Check_SINT_TO_BYTE_Min
VAR
	value : SINT := DatatypeLimits.MIN_VALUE_OF_SINT_WHICH_CAN_BE_HELD_IN_A_BYTE;
	actual : BYTE;
	converted : BOOL;
	equal : BOOL;
END_VAR
TEST('Check_SINT_TO_BYTE_Min');

// @TEST-RUN
converted := TryConvert_SINT_TO_Destination(value, actual);
equal := actual = SINT_TO_BYTE(value);

// @TEST-ASSERT
AssertTrue(Condition := equal, Message := 'Did not convert SINT to BYTE correctly');
AssertTrue(Condition := converted, Message := 'Did not report SINT to BYTE conversion was successful');

TEST_FINISHED();
END_METHOD

METHOD PUBLIC Check_SINT_TO_BYTE_TooLow
VAR
	value : SINT := DatatypeLimits.SINT_MIN_VALUE;
	actual : BYTE;
	converted : BOOL;
END_VAR
TEST('Check_SINT_TO_BYTE_TooLow');

// @TEST-RUN
converted := TryConvert_SINT_TO_Destination(value, actual);

// @TEST-ASSERT
AssertFalse(Condition := converted, Message := 'Did not report SINT to BYTE conversion was prevented');

TEST_FINISHED();
END_METHOD

METHOD PUBLIC Check_SINT_TO_BYTE_Max
VAR
	value : SINT := DatatypeLimits.SINT_MAX_VALUE;
	actual : BYTE;
	converted : BOOL;
	equal : BOOL;
END_VAR
TEST('Check_SINT_TO_BYTE_Max');

// @TEST-RUN
converted := TryConvert_SINT_TO_Destination(value, actual);
equal := actual = SINT_TO_BYTE(value);

// @TEST-ASSERT
AssertTrue(Condition := equal, Message := 'Did not convert SINT to BYTE correctly');
AssertTrue(Condition := converted, Message := 'Did not report SINT to BYTE conversion was successful');

TEST_FINISHED();
END_METHOD

METHOD PUBLIC Check_SINT_TO_DATE_Min
VAR
	value : SINT := DatatypeLimits.MIN_VALUE_OF_SINT_WHICH_CAN_BE_HELD_IN_A_DATE;
	actual : DATE;
	converted : BOOL;
	equal : BOOL;
END_VAR
TEST('Check_SINT_TO_DATE_Min');

// @TEST-RUN
converted := TryConvert_SINT_TO_Destination(value, actual);
equal := actual = SINT_TO_DATE(value);

// @TEST-ASSERT
AssertTrue(Condition := equal, Message := 'Did not convert SINT to DATE correctly');
AssertTrue(Condition := converted, Message := 'Did not report SINT to DATE conversion was successful');

TEST_FINISHED();
END_METHOD

METHOD PUBLIC Check_SINT_TO_DATE_TooLow
VAR
	value : SINT := DatatypeLimits.SINT_MIN_VALUE;
	actual : DATE;
	converted : BOOL;
END_VAR
TEST('Check_SINT_TO_DATE_TooLow');

// @TEST-RUN
converted := TryConvert_SINT_TO_Destination(value, actual);

// @TEST-ASSERT
AssertFalse(Condition := converted, Message := 'Did not report SINT to DATE conversion was prevented');

TEST_FINISHED();
END_METHOD

METHOD PUBLIC Check_SINT_TO_DATE_Max
VAR
	value : SINT := DatatypeLimits.SINT_MAX_VALUE;
	actual : DATE;
	converted : BOOL;
	equal : BOOL;
END_VAR
TEST('Check_SINT_TO_DATE_Max');

// @TEST-RUN
converted := TryConvert_SINT_TO_Destination(value, actual);
equal := actual = SINT_TO_DATE(value);

// @TEST-ASSERT
AssertTrue(Condition := equal, Message := 'Did not convert SINT to DATE correctly');
AssertTrue(Condition := converted, Message := 'Did not report SINT to DATE conversion was successful');

TEST_FINISHED();
END_METHOD

METHOD PUBLIC Check_SINT_TO_DINT_Min
VAR
	value : SINT := DatatypeLimits.SINT_MIN_VALUE;
	actual : DINT;
	converted : BOOL;
	equal : BOOL;
END_VAR
TEST('Check_SINT_TO_DINT_Min');

// @TEST-RUN
converted := TryConvert_SINT_TO_Destination(value, actual);
equal := actual = SINT_TO_DINT(value);

// @TEST-ASSERT
AssertTrue(Condition := equal, Message := 'Did not convert SINT to DINT correctly');
AssertTrue(Condition := converted, Message := 'Did not report SINT to DINT conversion was successful');

TEST_FINISHED();
END_METHOD

METHOD PUBLIC Check_SINT_TO_DINT_Max
VAR
	value : SINT := DatatypeLimits.SINT_MAX_VALUE;
	actual : DINT;
	converted : BOOL;
	equal : BOOL;
END_VAR
TEST('Check_SINT_TO_DINT_Max');

// @TEST-RUN
converted := TryConvert_SINT_TO_Destination(value, actual);
equal := actual = SINT_TO_DINT(value);

// @TEST-ASSERT
AssertTrue(Condition := equal, Message := 'Did not convert SINT to DINT correctly');
AssertTrue(Condition := converted, Message := 'Did not report SINT to DINT conversion was successful');

TEST_FINISHED();
END_METHOD

METHOD PUBLIC Check_SINT_TO_DT_Min
VAR
	value : SINT := DatatypeLimits.MIN_VALUE_OF_SINT_WHICH_CAN_BE_HELD_IN_A_DT;
	actual : DT;
	converted : BOOL;
	equal : BOOL;
END_VAR
TEST('Check_SINT_TO_DT_Min');

// @TEST-RUN
converted := TryConvert_SINT_TO_Destination(value, actual);
equal := actual = SINT_TO_DT(value);

// @TEST-ASSERT
AssertTrue(Condition := equal, Message := 'Did not convert SINT to DT correctly');
AssertTrue(Condition := converted, Message := 'Did not report SINT to DT conversion was successful');

TEST_FINISHED();
END_METHOD

METHOD PUBLIC Check_SINT_TO_DT_TooLow
VAR
	value : SINT := DatatypeLimits.SINT_MIN_VALUE;
	actual : DT;
	converted : BOOL;
END_VAR
TEST('Check_SINT_TO_DT_TooLow');

// @TEST-RUN
converted := TryConvert_SINT_TO_Destination(value, actual);

// @TEST-ASSERT
AssertFalse(Condition := converted, Message := 'Did not report SINT to DT conversion was prevented');

TEST_FINISHED();
END_METHOD

METHOD PUBLIC Check_SINT_TO_DT_Max
VAR
	value : SINT := DatatypeLimits.SINT_MAX_VALUE;
	actual : DT;
	converted : BOOL;
	equal : BOOL;
END_VAR
TEST('Check_SINT_TO_DT_Max');

// @TEST-RUN
converted := TryConvert_SINT_TO_Destination(value, actual);
equal := actual = SINT_TO_DT(value);

// @TEST-ASSERT
AssertTrue(Condition := equal, Message := 'Did not convert SINT to DT correctly');
AssertTrue(Condition := converted, Message := 'Did not report SINT to DT conversion was successful');

TEST_FINISHED();
END_METHOD

METHOD PUBLIC Check_SINT_TO_DWORD_Min
VAR
	value : SINT := DatatypeLimits.MIN_VALUE_OF_SINT_WHICH_CAN_BE_HELD_IN_A_DWORD;
	actual : DWORD;
	converted : BOOL;
	equal : BOOL;
END_VAR
TEST('Check_SINT_TO_DWORD_Min');

// @TEST-RUN
converted := TryConvert_SINT_TO_Destination(value, actual);
equal := actual = SINT_TO_DWORD(value);

// @TEST-ASSERT
AssertTrue(Condition := equal, Message := 'Did not convert SINT to DWORD correctly');
AssertTrue(Condition := converted, Message := 'Did not report SINT to DWORD conversion was successful');

TEST_FINISHED();
END_METHOD

METHOD PUBLIC Check_SINT_TO_DWORD_TooLow
VAR
	value : SINT := DatatypeLimits.SINT_MIN_VALUE;
	actual : DWORD;
	converted : BOOL;
END_VAR
TEST('Check_SINT_TO_DWORD_TooLow');

// @TEST-RUN
converted := TryConvert_SINT_TO_Destination(value, actual);

// @TEST-ASSERT
AssertFalse(Condition := converted, Message := 'Did not report SINT to DWORD conversion was prevented');

TEST_FINISHED();
END_METHOD

METHOD PUBLIC Check_SINT_TO_DWORD_Max
VAR
	value : SINT := DatatypeLimits.SINT_MAX_VALUE;
	actual : DWORD;
	converted : BOOL;
	equal : BOOL;
END_VAR
TEST('Check_SINT_TO_DWORD_Max');

// @TEST-RUN
converted := TryConvert_SINT_TO_Destination(value, actual);
equal := actual = SINT_TO_DWORD(value);

// @TEST-ASSERT
AssertTrue(Condition := equal, Message := 'Did not convert SINT to DWORD correctly');
AssertTrue(Condition := converted, Message := 'Did not report SINT to DWORD conversion was successful');

TEST_FINISHED();
END_METHOD

METHOD PUBLIC Check_SINT_TO_INT_Min
VAR
	value : SINT := DatatypeLimits.SINT_MIN_VALUE;
	actual : INT;
	converted : BOOL;
	equal : BOOL;
END_VAR
TEST('Check_SINT_TO_INT_Min');

// @TEST-RUN
converted := TryConvert_SINT_TO_Destination(value, actual);
equal := actual = SINT_TO_INT(value);

// @TEST-ASSERT
AssertTrue(Condition := equal, Message := 'Did not convert SINT to INT correctly');
AssertTrue(Condition := converted, Message := 'Did not report SINT to INT conversion was successful');

TEST_FINISHED();
END_METHOD

METHOD PUBLIC Check_SINT_TO_INT_Max
VAR
	value : SINT := DatatypeLimits.SINT_MAX_VALUE;
	actual : INT;
	converted : BOOL;
	equal : BOOL;
END_VAR
TEST('Check_SINT_TO_INT_Max');

// @TEST-RUN
converted := TryConvert_SINT_TO_Destination(value, actual);
equal := actual = SINT_TO_INT(value);

// @TEST-ASSERT
AssertTrue(Condition := equal, Message := 'Did not convert SINT to INT correctly');
AssertTrue(Condition := converted, Message := 'Did not report SINT to INT conversion was successful');

TEST_FINISHED();
END_METHOD

METHOD PUBLIC Check_SINT_TO_LINT_Min
VAR
	value : SINT := DatatypeLimits.SINT_MIN_VALUE;
	actual : LINT;
	converted : BOOL;
	equal : BOOL;
END_VAR
TEST('Check_SINT_TO_LINT_Min');

// @TEST-RUN
converted := TryConvert_SINT_TO_Destination(value, actual);
equal := actual = SINT_TO_LINT(value);

// @TEST-ASSERT
AssertTrue(Condition := equal, Message := 'Did not convert SINT to LINT correctly');
AssertTrue(Condition := converted, Message := 'Did not report SINT to LINT conversion was successful');

TEST_FINISHED();
END_METHOD

METHOD PUBLIC Check_SINT_TO_LINT_Max
VAR
	value : SINT := DatatypeLimits.SINT_MAX_VALUE;
	actual : LINT;
	converted : BOOL;
	equal : BOOL;
END_VAR
TEST('Check_SINT_TO_LINT_Max');

// @TEST-RUN
converted := TryConvert_SINT_TO_Destination(value, actual);
equal := actual = SINT_TO_LINT(value);

// @TEST-ASSERT
AssertTrue(Condition := equal, Message := 'Did not convert SINT to LINT correctly');
AssertTrue(Condition := converted, Message := 'Did not report SINT to LINT conversion was successful');

TEST_FINISHED();
END_METHOD

METHOD PUBLIC Check_SINT_TO_LREAL_Min
VAR
	value : SINT := DatatypeLimits.SINT_MIN_VALUE;
	actual : LREAL;
	converted : BOOL;
	equal : BOOL;
END_VAR
TEST('Check_SINT_TO_LREAL_Min');

// @TEST-RUN
converted := TryConvert_SINT_TO_Destination(value, actual);
equal := actual = SINT_TO_LREAL(value);

// @TEST-ASSERT
AssertTrue(Condition := equal, Message := 'Did not convert SINT to LREAL correctly');
AssertTrue(Condition := converted, Message := 'Did not report SINT to LREAL conversion was successful');

TEST_FINISHED();
END_METHOD

METHOD PUBLIC Check_SINT_TO_LREAL_Max
VAR
	value : SINT := DatatypeLimits.SINT_MAX_VALUE;
	actual : LREAL;
	converted : BOOL;
	equal : BOOL;
END_VAR
TEST('Check_SINT_TO_LREAL_Max');

// @TEST-RUN
converted := TryConvert_SINT_TO_Destination(value, actual);
equal := actual = SINT_TO_LREAL(value);

// @TEST-ASSERT
AssertTrue(Condition := equal, Message := 'Did not convert SINT to LREAL correctly');
AssertTrue(Condition := converted, Message := 'Did not report SINT to LREAL conversion was successful');

TEST_FINISHED();
END_METHOD

METHOD PUBLIC Check_SINT_TO_LWORD_Min
VAR
	value : SINT := DatatypeLimits.MIN_VALUE_OF_SINT_WHICH_CAN_BE_HELD_IN_A_LWORD;
	actual : LWORD;
	converted : BOOL;
	equal : BOOL;
END_VAR
TEST('Check_SINT_TO_LWORD_Min');

// @TEST-RUN
converted := TryConvert_SINT_TO_Destination(value, actual);
equal := actual = SINT_TO_LWORD(value);

// @TEST-ASSERT
AssertTrue(Condition := equal, Message := 'Did not convert SINT to LWORD correctly');
AssertTrue(Condition := converted, Message := 'Did not report SINT to LWORD conversion was successful');

TEST_FINISHED();
END_METHOD

METHOD PUBLIC Check_SINT_TO_LWORD_TooLow
VAR
	value : SINT := DatatypeLimits.SINT_MIN_VALUE;
	actual : LWORD;
	converted : BOOL;
END_VAR
TEST('Check_SINT_TO_LWORD_TooLow');

// @TEST-RUN
converted := TryConvert_SINT_TO_Destination(value, actual);

// @TEST-ASSERT
AssertFalse(Condition := converted, Message := 'Did not report SINT to LWORD conversion was prevented');

TEST_FINISHED();
END_METHOD

METHOD PUBLIC Check_SINT_TO_LWORD_Max
VAR
	value : SINT := DatatypeLimits.SINT_MAX_VALUE;
	actual : LWORD;
	converted : BOOL;
	equal : BOOL;
END_VAR
TEST('Check_SINT_TO_LWORD_Max');

// @TEST-RUN
converted := TryConvert_SINT_TO_Destination(value, actual);
equal := actual = SINT_TO_LWORD(value);

// @TEST-ASSERT
AssertTrue(Condition := equal, Message := 'Did not convert SINT to LWORD correctly');
AssertTrue(Condition := converted, Message := 'Did not report SINT to LWORD conversion was successful');

TEST_FINISHED();
END_METHOD

METHOD PUBLIC Check_SINT_TO_REAL_Min
VAR
	value : SINT := DatatypeLimits.SINT_MIN_VALUE;
	actual : REAL;
	converted : BOOL;
	equal : BOOL;
END_VAR
TEST('Check_SINT_TO_REAL_Min');

// @TEST-RUN
converted := TryConvert_SINT_TO_Destination(value, actual);
equal := actual = SINT_TO_REAL(value);

// @TEST-ASSERT
AssertTrue(Condition := equal, Message := 'Did not convert SINT to REAL correctly');
AssertTrue(Condition := converted, Message := 'Did not report SINT to REAL conversion was successful');

TEST_FINISHED();
END_METHOD

METHOD PUBLIC Check_SINT_TO_REAL_Max
VAR
	value : SINT := DatatypeLimits.SINT_MAX_VALUE;
	actual : REAL;
	converted : BOOL;
	equal : BOOL;
END_VAR
TEST('Check_SINT_TO_REAL_Max');

// @TEST-RUN
converted := TryConvert_SINT_TO_Destination(value, actual);
equal := actual = SINT_TO_REAL(value);

// @TEST-ASSERT
AssertTrue(Condition := equal, Message := 'Did not convert SINT to REAL correctly');
AssertTrue(Condition := converted, Message := 'Did not report SINT to REAL conversion was successful');

TEST_FINISHED();
END_METHOD

METHOD PUBLIC Check_SINT_TO_SINT_Min
VAR
	value : SINT := DatatypeLimits.SINT_MIN_VALUE;
	actual : SINT;
	converted : BOOL;
	equal : BOOL;
END_VAR
TEST('Check_SINT_TO_SINT_Min');

// @TEST-RUN
converted := TryConvert_SINT_TO_Destination(value, actual);
equal := actual = value;

// @TEST-ASSERT
AssertTrue(Condition := equal, Message := 'Did not convert SINT to SINT correctly');
AssertTrue(Condition := converted, Message := 'Did not report SINT to SINT conversion was successful');

TEST_FINISHED();
END_METHOD

METHOD PUBLIC Check_SINT_TO_SINT_Max
VAR
	value : SINT := DatatypeLimits.SINT_MAX_VALUE;
	actual : SINT;
	converted : BOOL;
	equal : BOOL;
END_VAR
TEST('Check_SINT_TO_SINT_Max');

// @TEST-RUN
converted := TryConvert_SINT_TO_Destination(value, actual);
equal := actual = value;

// @TEST-ASSERT
AssertTrue(Condition := equal, Message := 'Did not convert SINT to SINT correctly');
AssertTrue(Condition := converted, Message := 'Did not report SINT to SINT conversion was successful');

TEST_FINISHED();
END_METHOD

METHOD PUBLIC Check_SINT_TO_STRING_Min
VAR
	value : SINT := DatatypeLimits.SINT_MIN_VALUE;
	actual : STRING;
	converted : BOOL;
	equal : BOOL;
END_VAR
TEST('Check_SINT_TO_STRING_Min');

// @TEST-RUN
converted := TryConvert_SINT_TO_Destination(value, actual);
equal := actual = SINT_TO_STRING(value);

// @TEST-ASSERT
AssertTrue(Condition := equal, Message := 'Did not convert SINT to STRING correctly');
AssertTrue(Condition := converted, Message := 'Did not report SINT to STRING conversion was successful');

TEST_FINISHED();
END_METHOD

METHOD PUBLIC Check_SINT_TO_STRING_Max
VAR
	value : SINT := DatatypeLimits.SINT_MAX_VALUE;
	actual : STRING;
	converted : BOOL;
	equal : BOOL;
END_VAR
TEST('Check_SINT_TO_STRING_Max');

// @TEST-RUN
converted := TryConvert_SINT_TO_Destination(value, actual);
equal := actual = SINT_TO_STRING(value);

// @TEST-ASSERT
AssertTrue(Condition := equal, Message := 'Did not convert SINT to STRING correctly');
AssertTrue(Condition := converted, Message := 'Did not report SINT to STRING conversion was successful');

TEST_FINISHED();
END_METHOD

METHOD PUBLIC Check_SINT_TO_TIME_Min
VAR
	value : SINT := DatatypeLimits.MIN_VALUE_OF_SINT_WHICH_CAN_BE_HELD_IN_A_TIME;
	actual : TIME;
	converted : BOOL;
	equal : BOOL;
END_VAR
TEST('Check_SINT_TO_TIME_Min');

// @TEST-RUN
converted := TryConvert_SINT_TO_Destination(value, actual);
equal := actual = SINT_TO_TIME(value);

// @TEST-ASSERT
AssertTrue(Condition := equal, Message := 'Did not convert SINT to TIME correctly');
AssertTrue(Condition := converted, Message := 'Did not report SINT to TIME conversion was successful');

TEST_FINISHED();
END_METHOD

METHOD PUBLIC Check_SINT_TO_TIME_TooLow
VAR
	value : SINT := DatatypeLimits.SINT_MIN_VALUE;
	actual : TIME;
	converted : BOOL;
END_VAR
TEST('Check_SINT_TO_TIME_TooLow');

// @TEST-RUN
converted := TryConvert_SINT_TO_Destination(value, actual);

// @TEST-ASSERT
AssertFalse(Condition := converted, Message := 'Did not report SINT to TIME conversion was prevented');

TEST_FINISHED();
END_METHOD

METHOD PUBLIC Check_SINT_TO_TIME_Max
VAR
	value : SINT := DatatypeLimits.SINT_MAX_VALUE;
	actual : TIME;
	converted : BOOL;
	equal : BOOL;
END_VAR
TEST('Check_SINT_TO_TIME_Max');

// @TEST-RUN
converted := TryConvert_SINT_TO_Destination(value, actual);
equal := actual = SINT_TO_TIME(value);

// @TEST-ASSERT
AssertTrue(Condition := equal, Message := 'Did not convert SINT to TIME correctly');
AssertTrue(Condition := converted, Message := 'Did not report SINT to TIME conversion was successful');

TEST_FINISHED();
END_METHOD

METHOD PUBLIC Check_SINT_TO_TOD_Min
VAR
	value : SINT := DatatypeLimits.MIN_VALUE_OF_SINT_WHICH_CAN_BE_HELD_IN_A_TOD;
	actual : TOD;
	converted : BOOL;
	equal : BOOL;
END_VAR
TEST('Check_SINT_TO_TOD_Min');

// @TEST-RUN
converted := TryConvert_SINT_TO_Destination(value, actual);
equal := actual = SINT_TO_TOD(value);

// @TEST-ASSERT
AssertTrue(Condition := equal, Message := 'Did not convert SINT to TOD correctly');
AssertTrue(Condition := converted, Message := 'Did not report SINT to TOD conversion was successful');

TEST_FINISHED();
END_METHOD

METHOD PUBLIC Check_SINT_TO_TOD_TooLow
VAR
	value : SINT := DatatypeLimits.SINT_MIN_VALUE;
	actual : TOD;
	converted : BOOL;
END_VAR
TEST('Check_SINT_TO_TOD_TooLow');

// @TEST-RUN
converted := TryConvert_SINT_TO_Destination(value, actual);

// @TEST-ASSERT
AssertFalse(Condition := converted, Message := 'Did not report SINT to TOD conversion was prevented');

TEST_FINISHED();
END_METHOD

METHOD PUBLIC Check_SINT_TO_TOD_Max
VAR
	value : SINT := DatatypeLimits.SINT_MAX_VALUE;
	actual : TOD;
	converted : BOOL;
	equal : BOOL;
END_VAR
TEST('Check_SINT_TO_TOD_Max');

// @TEST-RUN
converted := TryConvert_SINT_TO_Destination(value, actual);
equal := actual = SINT_TO_TOD(value);

// @TEST-ASSERT
AssertTrue(Condition := equal, Message := 'Did not convert SINT to TOD correctly');
AssertTrue(Condition := converted, Message := 'Did not report SINT to TOD conversion was successful');

TEST_FINISHED();
END_METHOD

METHOD PUBLIC Check_SINT_TO_UDINT_Min
VAR
	value : SINT := DatatypeLimits.MIN_VALUE_OF_SINT_WHICH_CAN_BE_HELD_IN_A_UDINT;
	actual : UDINT;
	converted : BOOL;
	equal : BOOL;
END_VAR
TEST('Check_SINT_TO_UDINT_Min');

// @TEST-RUN
converted := TryConvert_SINT_TO_Destination(value, actual);
equal := actual = SINT_TO_UDINT(value);

// @TEST-ASSERT
AssertTrue(Condition := equal, Message := 'Did not convert SINT to UDINT correctly');
AssertTrue(Condition := converted, Message := 'Did not report SINT to UDINT conversion was successful');

TEST_FINISHED();
END_METHOD

METHOD PUBLIC Check_SINT_TO_UDINT_TooLow
VAR
	value : SINT := DatatypeLimits.SINT_MIN_VALUE;
	actual : UDINT;
	converted : BOOL;
END_VAR
TEST('Check_SINT_TO_UDINT_TooLow');

// @TEST-RUN
converted := TryConvert_SINT_TO_Destination(value, actual);

// @TEST-ASSERT
AssertFalse(Condition := converted, Message := 'Did not report SINT to UDINT conversion was prevented');

TEST_FINISHED();
END_METHOD

METHOD PUBLIC Check_SINT_TO_UDINT_Max
VAR
	value : SINT := DatatypeLimits.SINT_MAX_VALUE;
	actual : UDINT;
	converted : BOOL;
	equal : BOOL;
END_VAR
TEST('Check_SINT_TO_UDINT_Max');

// @TEST-RUN
converted := TryConvert_SINT_TO_Destination(value, actual);
equal := actual = SINT_TO_UDINT(value);

// @TEST-ASSERT
AssertTrue(Condition := equal, Message := 'Did not convert SINT to UDINT correctly');
AssertTrue(Condition := converted, Message := 'Did not report SINT to UDINT conversion was successful');

TEST_FINISHED();
END_METHOD

METHOD PUBLIC Check_SINT_TO_UINT_Min
VAR
	value : SINT := DatatypeLimits.MIN_VALUE_OF_SINT_WHICH_CAN_BE_HELD_IN_A_UINT;
	actual : UINT;
	converted : BOOL;
	equal : BOOL;
END_VAR
TEST('Check_SINT_TO_UINT_Min');

// @TEST-RUN
converted := TryConvert_SINT_TO_Destination(value, actual);
equal := actual = SINT_TO_UINT(value);

// @TEST-ASSERT
AssertTrue(Condition := equal, Message := 'Did not convert SINT to UINT correctly');
AssertTrue(Condition := converted, Message := 'Did not report SINT to UINT conversion was successful');

TEST_FINISHED();
END_METHOD

METHOD PUBLIC Check_SINT_TO_UINT_TooLow
VAR
	value : SINT := DatatypeLimits.SINT_MIN_VALUE;
	actual : UINT;
	converted : BOOL;
END_VAR
TEST('Check_SINT_TO_UINT_TooLow');

// @TEST-RUN
converted := TryConvert_SINT_TO_Destination(value, actual);

// @TEST-ASSERT
AssertFalse(Condition := converted, Message := 'Did not report SINT to UINT conversion was prevented');

TEST_FINISHED();
END_METHOD

METHOD PUBLIC Check_SINT_TO_UINT_Max
VAR
	value : SINT := DatatypeLimits.SINT_MAX_VALUE;
	actual : UINT;
	converted : BOOL;
	equal : BOOL;
END_VAR
TEST('Check_SINT_TO_UINT_Max');

// @TEST-RUN
converted := TryConvert_SINT_TO_Destination(value, actual);
equal := actual = SINT_TO_UINT(value);

// @TEST-ASSERT
AssertTrue(Condition := equal, Message := 'Did not convert SINT to UINT correctly');
AssertTrue(Condition := converted, Message := 'Did not report SINT to UINT conversion was successful');

TEST_FINISHED();
END_METHOD

METHOD PUBLIC Check_SINT_TO_ULINT_Min
VAR
	value : SINT := DatatypeLimits.MIN_VALUE_OF_SINT_WHICH_CAN_BE_HELD_IN_A_ULINT;
	actual : ULINT;
	converted : BOOL;
	equal : BOOL;
END_VAR
TEST('Check_SINT_TO_ULINT_Min');

// @TEST-RUN
converted := TryConvert_SINT_TO_Destination(value, actual);
equal := actual = SINT_TO_ULINT(value);

// @TEST-ASSERT
AssertTrue(Condition := equal, Message := 'Did not convert SINT to ULINT correctly');
AssertTrue(Condition := converted, Message := 'Did not report SINT to ULINT conversion was successful');

TEST_FINISHED();
END_METHOD

METHOD PUBLIC Check_SINT_TO_ULINT_TooLow
VAR
	value : SINT := DatatypeLimits.SINT_MIN_VALUE;
	actual : ULINT;
	converted : BOOL;
END_VAR
TEST('Check_SINT_TO_ULINT_TooLow');

// @TEST-RUN
converted := TryConvert_SINT_TO_Destination(value, actual);

// @TEST-ASSERT
AssertFalse(Condition := converted, Message := 'Did not report SINT to ULINT conversion was prevented');

TEST_FINISHED();
END_METHOD

METHOD PUBLIC Check_SINT_TO_ULINT_Max
VAR
	value : SINT := DatatypeLimits.SINT_MAX_VALUE;
	actual : ULINT;
	converted : BOOL;
	equal : BOOL;
END_VAR
TEST('Check_SINT_TO_ULINT_Max');

// @TEST-RUN
converted := TryConvert_SINT_TO_Destination(value, actual);
equal := actual = SINT_TO_ULINT(value);

// @TEST-ASSERT
AssertTrue(Condition := equal, Message := 'Did not convert SINT to ULINT correctly');
AssertTrue(Condition := converted, Message := 'Did not report SINT to ULINT conversion was successful');

TEST_FINISHED();
END_METHOD

METHOD PUBLIC Check_SINT_TO_USINT_Min
VAR
	value : SINT := DatatypeLimits.MIN_VALUE_OF_SINT_WHICH_CAN_BE_HELD_IN_A_USINT;
	actual : USINT;
	converted : BOOL;
	equal : BOOL;
END_VAR
TEST('Check_SINT_TO_USINT_Min');

// @TEST-RUN
converted := TryConvert_SINT_TO_Destination(value, actual);
equal := actual = SINT_TO_USINT(value);

// @TEST-ASSERT
AssertTrue(Condition := equal, Message := 'Did not convert SINT to USINT correctly');
AssertTrue(Condition := converted, Message := 'Did not report SINT to USINT conversion was successful');

TEST_FINISHED();
END_METHOD

METHOD PUBLIC Check_SINT_TO_USINT_TooLow
VAR
	value : SINT := DatatypeLimits.SINT_MIN_VALUE;
	actual : USINT;
	converted : BOOL;
END_VAR
TEST('Check_SINT_TO_USINT_TooLow');

// @TEST-RUN
converted := TryConvert_SINT_TO_Destination(value, actual);

// @TEST-ASSERT
AssertFalse(Condition := converted, Message := 'Did not report SINT to USINT conversion was prevented');

TEST_FINISHED();
END_METHOD

METHOD PUBLIC Check_SINT_TO_USINT_Max
VAR
	value : SINT := DatatypeLimits.SINT_MAX_VALUE;
	actual : USINT;
	converted : BOOL;
	equal : BOOL;
END_VAR
TEST('Check_SINT_TO_USINT_Max');

// @TEST-RUN
converted := TryConvert_SINT_TO_Destination(value, actual);
equal := actual = SINT_TO_USINT(value);

// @TEST-ASSERT
AssertTrue(Condition := equal, Message := 'Did not convert SINT to USINT correctly');
AssertTrue(Condition := converted, Message := 'Did not report SINT to USINT conversion was successful');

TEST_FINISHED();
END_METHOD

METHOD PUBLIC Check_SINT_TO_WORD_Min
VAR
	value : SINT := DatatypeLimits.MIN_VALUE_OF_SINT_WHICH_CAN_BE_HELD_IN_A_WORD;
	actual : WORD;
	converted : BOOL;
	equal : BOOL;
END_VAR
TEST('Check_SINT_TO_WORD_Min');

// @TEST-RUN
converted := TryConvert_SINT_TO_Destination(value, actual);
equal := actual = SINT_TO_WORD(value);

// @TEST-ASSERT
AssertTrue(Condition := equal, Message := 'Did not convert SINT to WORD correctly');
AssertTrue(Condition := converted, Message := 'Did not report SINT to WORD conversion was successful');

TEST_FINISHED();
END_METHOD

METHOD PUBLIC Check_SINT_TO_WORD_TooLow
VAR
	value : SINT := DatatypeLimits.SINT_MIN_VALUE;
	actual : WORD;
	converted : BOOL;
END_VAR
TEST('Check_SINT_TO_WORD_TooLow');

// @TEST-RUN
converted := TryConvert_SINT_TO_Destination(value, actual);

// @TEST-ASSERT
AssertFalse(Condition := converted, Message := 'Did not report SINT to WORD conversion was prevented');

TEST_FINISHED();
END_METHOD

METHOD PUBLIC Check_SINT_TO_WORD_Max
VAR
	value : SINT := DatatypeLimits.SINT_MAX_VALUE;
	actual : WORD;
	converted : BOOL;
	equal : BOOL;
END_VAR
TEST('Check_SINT_TO_WORD_Max');

// @TEST-RUN
converted := TryConvert_SINT_TO_Destination(value, actual);
equal := actual = SINT_TO_WORD(value);

// @TEST-ASSERT
AssertTrue(Condition := equal, Message := 'Did not convert SINT to WORD correctly');
AssertTrue(Condition := converted, Message := 'Did not report SINT to WORD conversion was successful');

TEST_FINISHED();
END_METHOD

END_FUNCTION_BLOCK

// ---- Tests/INT_TO_TestSuite.TcPOU
FUNCTION_BLOCK PUBLIC INT_TO_TestSuite EXTENDS TcUnit.FB_TestSuite
VAR
END_VAR

Check_INT_TO_BOOL_Max();
Check_INT_TO_BOOL_Min();
Check_INT_TO_BYTE_Max();
Check_INT_TO_BYTE_Min();
Check_INT_TO_BYTE_TooHigh();
Check_INT_TO_BYTE_TooLow();
Check_INT_TO_WORD_Max();
Check_INT_TO_WORD_Min();
Check_INT_TO_WORD_TooLow();
Check_INT_TO_DWORD_Max();
Check_INT_TO_DWORD_Min();
Check_INT_TO_DWORD_TooLow();
Check_INT_TO_LWORD_Max();
Check_INT_TO_LWORD_Min();
Check_INT_TO_LWORD_TooLow();
Check_INT_TO_SINT_Max();
Check_INT_TO_SINT_Min();
Check_INT_TO_SINT_TooHigh();
Check_INT_TO_SINT_TooLow();
Check_INT_TO_INT_Max();
Check_INT_TO_INT_Min();
Check_INT_TO_DINT_Max();
Check_INT_TO_DINT_Min();
Check_INT_TO_LINT_Max();
Check_INT_TO_LINT_Min();
Check_INT_TO_USINT_Max();
Check_INT_TO_USINT_Min();
Check_INT_TO_USINT_TooHigh();
Check_INT_TO_USINT_TooLow();
Check_INT_TO_UINT_Max();
Check_INT_TO_UINT_Min();
Check_INT_TO_UINT_TooLow();
Check_INT_TO_UDINT_Max();
Check_INT_TO_UDINT_Min();
Check_INT_TO_UDINT_TooLow();
Check_INT_TO_ULINT_Max();
Check_INT_TO_ULINT_Min();
Check_INT_TO_ULINT_TooLow();
Check_INT_TO_REAL_Max();
Check_INT_TO_REAL_Min();
Check_INT_TO_LREAL_Max();
Check_INT_TO_LREAL_Min();
Check_INT_TO_TIME_Max();
Check_INT_TO_TIME_Min();
Check_INT_TO_TIME_TooLow();
Check_INT_TO_TOD_Max();
Check_INT_TO_TOD_Min();
Check_INT_TO_TOD_TooLow();
Check_INT_TO_DATE_Max();
Check_INT_TO_DATE_Min();
Check_INT_TO_DATE_TooLow();
Check_INT_TO_DT_Max();
Check_INT_TO_DT_Min();
Check_INT_TO_DT_TooLow();
Check_INT_TO_STRING_Max();
Check_INT_TO_STRING_Min();

METHOD PUBLIC Check_INT_TO_BOOL_Min
VAR
	value : INT := DatatypeLimits.INT_MIN_VALUE;
	actual : BOOL;
	converted : BOOL;
	equal : BOOL;
END_VAR
TEST('Check_INT_TO_BOOL_Min');

// @TEST-RUN
converted := TryConvert_INT_TO_Destination(value, actual);
equal := actual = INT_TO_BOOL(value);

// @TEST-ASSERT
AssertTrue(Condition := equal, Message := 'Did not convert INT to BOOL correctly');
AssertTrue(Condition := converted, Message := 'Did not report INT to BOOL conversion was successful');

TEST_FINISHED();
END_METHOD

METHOD PUBLIC Check_INT_TO_BOOL_Max
VAR
	value : INT := DatatypeLimits.INT_MAX_VALUE;
	actual : BOOL;
	converted : BOOL;
	equal : BOOL;
END_VAR
TEST('Check_INT_TO_BOOL_Max');

// @TEST-RUN
converted := TryConvert_INT_TO_Destination(value, actual);
equal := actual = INT_TO_BOOL(value);

// @TEST-ASSERT
AssertTrue(Condition := equal, Message := 'Did not convert INT to BOOL correctly');
AssertTrue(Condition := converted, Message := 'Did not report INT to BOOL conversion was successful');

TEST_FINISHED();
END_METHOD

METHOD PUBLIC Check_INT_TO_BYTE_Min
VAR
	value : INT := DatatypeLimits.MIN_VALUE_OF_INT_WHICH_CAN_BE_HELD_IN_A_BYTE;
	actual : BYTE;
	converted : BOOL;
	equal : BOOL;
END_VAR
TEST('Check_INT_TO_BYTE_Min');

// @TEST-RUN
converted := TryConvert_INT_TO_Destination(value, actual);
equal := actual = INT_TO_BYTE(value);

// @TEST-ASSERT
AssertTrue(Condition := equal, Message := 'Did not convert INT to BYTE correctly');
AssertTrue(Condition := converted, Message := 'Did not report INT to BYTE conversion was successful');

TEST_FINISHED();
END_METHOD

METHOD PUBLIC Check_INT_TO_BYTE_TooHigh
VAR
	value : INT := DatatypeLimits.INT_MAX_VALUE;
	actual : BYTE;
	converted : BOOL;
END_VAR
TEST('Check_INT_TO_BYTE_TooHigh');

// @TEST-RUN
converted := TryConvert_INT_TO_Destination(value, actual);

// @TEST-ASSERT
AssertFalse(Condition := converted, Message := 'Did not report INT to BYTE conversion was prevented');

TEST_FINISHED();
END_METHOD

METHOD PUBLIC Check_INT_TO_BYTE_TooLow
VAR
	value : INT := DatatypeLimits.INT_MIN_VALUE;
	actual : BYTE;
	converted : BOOL;
END_VAR
TEST('Check_INT_TO_BYTE_TooLow');

// @TEST-RUN
converted := TryConvert_INT_TO_Destination(value, actual);

// @TEST-ASSERT
AssertFalse(Condition := converted, Message := 'Did not report INT to BYTE conversion was prevented');

TEST_FINISHED();
END_METHOD

METHOD PUBLIC Check_INT_TO_BYTE_Max
VAR
	value : INT := DatatypeLimits.MAX_VALUE_OF_INT_WHICH_CAN_BE_HELD_IN_A_BYTE;
	actual : BYTE;
	converted : BOOL;
	equal : BOOL;
END_VAR
TEST('Check_INT_TO_BYTE_Max');

// @TEST-RUN
converted := TryConvert_INT_TO_Destination(value, actual);
equal := actual = INT_TO_BYTE(value);

// @TEST-ASSERT
AssertTrue(Condition := equal, Message := 'Did not convert INT to BYTE correctly');
AssertTrue(Condition := converted, Message := 'Did not report INT to BYTE conversion was successful');

TEST_FINISHED();
END_METHOD

METHOD PUBLIC Check_INT_TO_DATE_Min
VAR
	value : INT := DatatypeLimits.MIN_VALUE_OF_INT_WHICH_CAN_BE_HELD_IN_A_DATE;
	actual : DATE;
	converted : BOOL;
	equal : BOOL;
END_VAR
TEST('Check_INT_TO_DATE_Min');

// @TEST-RUN
converted := TryConvert_INT_TO_Destination(value, actual);
equal := actual = INT_TO_DATE(value);

// @TEST-ASSERT
AssertTrue(Condition := equal, Message := 'Did not convert INT to DATE correctly');
AssertTrue(Condition := converted, Message := 'Did not report INT to DATE conversion was successful');

TEST_FINISHED();
END_METHOD

METHOD PUBLIC Check_INT_TO_DATE_TooLow
VAR
	value : INT := DatatypeLimits.INT_MIN_VALUE;
	actual : DATE;
	converted : BOOL;
END_VAR
TEST('Check_INT_TO_DATE_TooLow');

// @TEST-RUN
converted := TryConvert_INT_TO_Destination(value, actual);

// @TEST-ASSERT
AssertFalse(Condition := converted, Message := 'Did not report INT to DATE conversion was prevented');

TEST_FINISHED();
END_METHOD

METHOD PUBLIC Check_INT_TO_DATE_Max
VAR
	value : INT := DatatypeLimits.INT_MAX_VALUE;
	actual : DATE;
	converted : BOOL;
	equal : BOOL;
END_VAR
TEST('Check_INT_TO_DATE_Max');

// @TEST-RUN
converted := TryConvert_INT_TO_Destination(value, actual);
equal := actual = INT_TO_DATE(value);

// @TEST-ASSERT
AssertTrue(Condition := equal, Message := 'Did not convert INT to DATE correctly');
AssertTrue(Condition := converted, Message := 'Did not report INT to DATE conversion was successful');

TEST_FINISHED();
END_METHOD

METHOD PUBLIC Check_INT_TO_DINT_Min
VAR
	value : INT := DatatypeLimits.INT_MIN_VALUE;
	actual : DINT;
	converted : BOOL;
	equal : BOOL;
END_VAR
TEST('Check_INT_TO_DINT_Min');

// @TEST-RUN
converted := TryConvert_INT_TO_Destination(value, actual);
equal := actual = INT_TO_DINT(value);

// @TEST-ASSERT
AssertTrue(Condition := equal, Message := 'Did not convert INT to DINT correctly');
AssertTrue(Condition := converted, Message := 'Did not report INT to DINT conversion was successful');

TEST_FINISHED();
END_METHOD

METHOD PUBLIC Check_INT_TO_DINT_Max
VAR
	value : INT := DatatypeLimits.INT_MAX_VALUE;
	actual : DINT;
	converted : BOOL;
	equal : BOOL;
END_VAR
TEST('Check_INT_TO_DINT_Max');

// @TEST-RUN
converted := TryConvert_INT_TO_Destination(value, actual);
equal := actual = INT_TO_DINT(value);

// @TEST-ASSERT
AssertTrue(Condition := equal, Message := 'Did not convert INT to DINT correctly');
AssertTrue(Condition := converted, Message := 'Did not report INT to DINT conversion was successful');

TEST_FINISHED();
END_METHOD

METHOD PUBLIC Check_INT_TO_DT_Min
VAR
	value : INT := DatatypeLimits.MIN_VALUE_OF_INT_WHICH_CAN_BE_HELD_IN_A_DT;
	actual : DT;
	converted : BOOL;
	equal : BOOL;
END_VAR
TEST('Check_INT_TO_DT_Min');

// @TEST-RUN
converted := TryConvert_INT_TO_Destination(value, actual);
equal := actual = INT_TO_DT(value);

// @TEST-ASSERT
AssertTrue(Condition := equal, Message := 'Did not convert INT to DT correctly');
AssertTrue(Condition := converted, Message := 'Did not report INT to DT conversion was successful');

TEST_FINISHED();
END_METHOD

METHOD PUBLIC Check_INT_TO_DT_TooLow
VAR
	value : INT := DatatypeLimits.INT_MIN_VALUE;
	actual : DT;
	converted : BOOL;
END_VAR
TEST('Check_INT_TO_DT_TooLow');

// @TEST-RUN
converted := TryConvert_INT_TO_Destination(value, actual);

// @TEST-ASSERT
AssertFalse(Condition := converted, Message := 'Did not report INT to DT conversion was prevented');

TEST_FINISHED();
END_METHOD

METHOD PUBLIC Check_INT_TO_DT_Max
VAR
	value : INT := DatatypeLimits.INT_MAX_VALUE;
	actual : DT;
	converted : BOOL;
	equal : BOOL;
END_VAR
TEST('Check_INT_TO_DT_Max');

// @TEST-RUN
converted := TryConvert_INT_TO_Destination(value, actual);
equal := actual = INT_TO_DT(value);

// @TEST-ASSERT
AssertTrue(Condition := equal, Message := 'Did not convert INT to DT correctly');
AssertTrue(Condition := converted, Message := 'Did not report INT to DT conversion was successful');

TEST_FINISHED();
END_METHOD

METHOD PUBLIC Check_INT_TO_DWORD_Min
VAR
	value : INT := DatatypeLimits.MIN_VALUE_OF_INT_WHICH_CAN_BE_HELD_IN_A_DWORD;
	actual : DWORD;
	converted : BOOL;
	equal : BOOL;
END_VAR
TEST('Check_INT_TO_DWORD_Min');

// @TEST-RUN
converted := TryConvert_INT_TO_Destination(value, actual);
equal := actual = INT_TO_DWORD(value);

// @TEST-ASSERT
AssertTrue(Condition := equal, Message := 'Did not convert INT to DWORD correctly');
AssertTrue(Condition := converted, Message := 'Did not report INT to DWORD conversion was successful');

TEST_FINISHED();
END_METHOD

METHOD PUBLIC Check_INT_TO_DWORD_TooLow
VAR
	value : INT := DatatypeLimits.INT_MIN_VALUE;
	actual : DWORD;
	converted : BOOL;
END_VAR
TEST('Check_INT_TO_DWORD_TooLow');

// @TEST-RUN
converted := TryConvert_INT_TO_Destination(value, actual);

// @TEST-ASSERT
AssertFalse(Condition := converted, Message := 'Did not report INT to DWORD conversion was prevented');

TEST_FINISHED();
END_METHOD

METHOD PUBLIC Check_INT_TO_DWORD_Max
VAR
	value : INT := DatatypeLimits.INT_MAX_VALUE;
	actual : DWORD;
	converted : BOOL;
	equal : BOOL;
END_VAR
TEST('Check_INT_TO_DWORD_Max');

// @TEST-RUN
converted := TryConvert_INT_TO_Destination(value, actual);
equal := actual = INT_TO_DWORD(value);

// @TEST-ASSERT
AssertTrue(Condition := equal, Message := 'Did not convert INT to DWORD correctly');
AssertTrue(Condition := converted, Message := 'Did not report INT to DWORD conversion was successful');

TEST_FINISHED();
END_METHOD

METHOD PUBLIC Check_INT_TO_INT_Min
VAR
	value : INT := DatatypeLimits.INT_MIN_VALUE;
	actual : INT;
	converted : BOOL;
	equal : BOOL;
END_VAR
TEST('Check_INT_TO_INT_Min');

// @TEST-RUN
converted := TryConvert_INT_TO_Destination(value, actual);
equal := actual = value;

// @TEST-ASSERT
AssertTrue(Condition := equal, Message := 'Did not convert INT to INT correctly');
AssertTrue(Condition := converted, Message := 'Did not report INT to INT conversion was successful');

TEST_FINISHED();
END_METHOD

METHOD PUBLIC Check_INT_TO_INT_Max
VAR
	value : INT := DatatypeLimits.INT_MAX_VALUE;
	actual : INT;
	converted : BOOL;
	equal : BOOL;
END_VAR
TEST('Check_INT_TO_INT_Max');

// @TEST-RUN
converted := TryConvert_INT_TO_Destination(value, actual);
equal := actual = value;

// @TEST-ASSERT
AssertTrue(Condition := equal, Message := 'Did not convert INT to INT correctly');
AssertTrue(Condition := converted, Message := 'Did not report INT to INT conversion was successful');

TEST_FINISHED();
END_METHOD

METHOD PUBLIC Check_INT_TO_LINT_Min
VAR
	value : INT := DatatypeLimits.INT_MIN_VALUE;
	actual : LINT;
	converted : BOOL;
	equal : BOOL;
END_VAR
TEST('Check_INT_TO_LINT_Min');

// @TEST-RUN
converted := TryConvert_INT_TO_Destination(value, actual);
equal := actual = INT_TO_LINT(value);

// @TEST-ASSERT
AssertTrue(Condition := equal, Message := 'Did not convert INT to LINT correctly');
AssertTrue(Condition := converted, Message := 'Did not report INT to LINT conversion was successful');

TEST_FINISHED();
END_METHOD

METHOD PUBLIC Check_INT_TO_LINT_Max
VAR
	value : INT := DatatypeLimits.INT_MAX_VALUE;
	actual : LINT;
	converted : BOOL;
	equal : BOOL;
END_VAR
TEST('Check_INT_TO_LINT_Max');

// @TEST-RUN
converted := TryConvert_INT_TO_Destination(value, actual);
equal := actual = INT_TO_LINT(value);

// @TEST-ASSERT
AssertTrue(Condition := equal, Message := 'Did not convert INT to LINT correctly');
AssertTrue(Condition := converted, Message := 'Did not report INT to LINT conversion was successful');

TEST_FINISHED();
END_METHOD

METHOD PUBLIC Check_INT_TO_LREAL_Min
VAR
	value : INT := DatatypeLimits.INT_MIN_VALUE;
	actual : LREAL;
	converted : BOOL;
	equal : BOOL;
END_VAR
TEST('Check_INT_TO_LREAL_Min');

// @TEST-RUN
converted := TryConvert_INT_TO_Destination(value, actual);
equal := actual = INT_TO_LREAL(value);

// @TEST-ASSERT
AssertTrue(Condition := equal, Message := 'Did not convert INT to LREAL correctly');
AssertTrue(Condition := converted, Message := 'Did not report INT to LREAL conversion was successful');

TEST_FINISHED();
END_METHOD

METHOD PUBLIC Check_INT_TO_LREAL_Max
VAR
	value : INT := DatatypeLimits.INT_MAX_VALUE;
	actual : LREAL;
	converted : BOOL;
	equal : BOOL;
END_VAR
TEST('Check_INT_TO_LREAL_Max');

// @TEST-RUN
converted := TryConvert_INT_TO_Destination(value, actual);
equal := actual = INT_TO_LREAL(value);

// @TEST-ASSERT
AssertTrue(Condition := equal, Message := 'Did not convert INT to LREAL correctly');
AssertTrue(Condition := converted, Message := 'Did not report INT to LREAL conversion was successful');

TEST_FINISHED();
END_METHOD

METHOD PUBLIC Check_INT_TO_LWORD_Min
VAR
	value : INT := DatatypeLimits.MIN_VALUE_OF_INT_WHICH_CAN_BE_HELD_IN_A_LWORD;
	actual : LWORD;
	converted : BOOL;
	equal : BOOL;
END_VAR
TEST('Check_INT_TO_LWORD_Min');

// @TEST-RUN
converted := TryConvert_INT_TO_Destination(value, actual);
equal := actual = INT_TO_LWORD(value);

// @TEST-ASSERT
AssertTrue(Condition := equal, Message := 'Did not convert INT to LWORD correctly');
AssertTrue(Condition := converted, Message := 'Did not report INT to LWORD conversion was successful');

TEST_FINISHED();
END_METHOD

METHOD PUBLIC Check_INT_TO_LWORD_TooLow
VAR
	value : INT := DatatypeLimits.INT_MIN_VALUE;
	actual : LWORD;
	converted : BOOL;
END_VAR
TEST('Check_INT_TO_LWORD_TooLow');

// @TEST-RUN
converted := TryConvert_INT_TO_Destination(value, actual);

// @TEST-ASSERT
AssertFalse(Condition := converted, Message := 'Did not report INT to LWORD conversion was prevented');

TEST_FINISHED();
END_METHOD

METHOD PUBLIC Check_INT_TO_LWORD_Max
VAR
	value : INT := DatatypeLimits.INT_MAX_VALUE;
	actual : LWORD;
	converted : BOOL;
	equal : BOOL;
END_VAR
TEST('Check_INT_TO_LWORD_Max');

// @TEST-RUN
converted := TryConvert_INT_TO_Destination(value, actual);
equal := actual = INT_TO_LWORD(value);

// @TEST-ASSERT
AssertTrue(Condition := equal, Message := 'Did not convert INT to LWORD correctly');
AssertTrue(Condition := converted, Message := 'Did not report INT to LWORD conversion was successful');

TEST_FINISHED();
END_METHOD

METHOD PUBLIC Check_INT_TO_REAL_Min
VAR
	value : INT := DatatypeLimits.INT_MIN_VALUE;
	actual : REAL;
	converted : BOOL;
	equal : BOOL;
END_VAR
TEST('Check_INT_TO_REAL_Min');

// @TEST-RUN
converted := TryConvert_INT_TO_Destination(value, actual);
equal := actual = INT_TO_REAL(value);

// @TEST-ASSERT
AssertTrue(Condition := equal, Message := 'Did not convert INT to REAL correctly');
AssertTrue(Condition := converted, Message := 'Did not report INT to REAL conversion was successful');

TEST_FINISHED();
END_METHOD

METHOD PUBLIC Check_INT_TO_REAL_Max
VAR
	value : INT := DatatypeLimits.INT_MAX_VALUE;
	actual : REAL;
	converted : BOOL;
	equal : BOOL;
END_VAR
TEST('Check_INT_TO_REAL_Max');

// @TEST-RUN
converted := TryConvert_INT_TO_Destination(value, actual);
equal := actual = INT_TO_REAL(value);

// @TEST-ASSERT
AssertTrue(Condition := equal, Message := 'Did not convert INT to REAL correctly');
AssertTrue(Condition := converted, Message := 'Did not report INT to REAL conversion was successful');

TEST_FINISHED();
END_METHOD

METHOD PUBLIC Check_INT_TO_SINT_Min
VAR
	value : INT := DatatypeLimits.MIN_VALUE_OF_INT_WHICH_CAN_BE_HELD_IN_A_SINT;
	actual : SINT;
	converted : BOOL;
	equal : BOOL;
END_VAR
TEST('Check_INT_TO_SINT_Min');

// @TEST-RUN
converted := TryConvert_INT_TO_Destination(value, actual);
equal := actual = INT_TO_SINT(value);

// @TEST-ASSERT
AssertTrue(Condition := equal, Message := 'Did not convert INT to SINT correctly');
AssertTrue(Condition := converted, Message := 'Did not report INT to SINT conversion was successful');

TEST_FINISHED();
END_METHOD

METHOD PUBLIC Check_INT_TO_SINT_TooHigh
VAR
	value : INT := DatatypeLimits.INT_MAX_VALUE;
	actual : SINT;
	converted : BOOL;
END_VAR
TEST('Check_INT_TO_SINT_TooHigh');

// @TEST-RUN
converted := TryConvert_INT_TO_Destination(value, actual);

// @TEST-ASSERT
AssertFalse(Condition := converted, Message := 'Did not report INT to SINT conversion was prevented');

TEST_FINISHED();
END_METHOD

METHOD PUBLIC Check_INT_TO_SINT_TooLow
VAR
	value : INT := DatatypeLimits.INT_MIN_VALUE;
	actual : SINT;
	converted : BOOL;
END_VAR
TEST('Check_INT_TO_SINT_TooLow');

// @TEST-RUN
converted := TryConvert_INT_TO_Destination(value, actual);

// @TEST-ASSERT
AssertFalse(Condition := converted, Message := 'Did not report INT to SINT conversion was prevented');

TEST_FINISHED();
END_METHOD

METHOD PUBLIC Check_INT_TO_SINT_Max
VAR
	value : INT := DatatypeLimits.MAX_VALUE_OF_INT_WHICH_CAN_BE_HELD_IN_A_SINT;
	actual : SINT;
	converted : BOOL;
	equal : BOOL;
END_VAR
TEST('Check_INT_TO_SINT_Max');

// @TEST-RUN
converted := TryConvert_INT_TO_Destination(value, actual);
equal := actual = INT_TO_SINT(value);

// @TEST-ASSERT
AssertTrue(Condition := equal, Message := 'Did not convert INT to SINT correctly');
AssertTrue(Condition := converted, Message := 'Did not report INT to SINT conversion was successful');

TEST_FINISHED();
END_METHOD

METHOD PUBLIC Check_INT_TO_STRING_Min
VAR
	value : INT := DatatypeLimits.INT_MIN_VALUE;
	actual : STRING;
	converted : BOOL;
	equal : BOOL;
END_VAR
TEST('Check_INT_TO_STRING_Min');

// @TEST-RUN
converted := TryConvert_INT_TO_Destination(value, actual);
equal := actual = INT_TO_STRING(value);

// @TEST-ASSERT
AssertTrue(Condition := equal, Message := 'Did not convert INT to STRING correctly');
AssertTrue(Condition := converted, Message := 'Did not report INT to STRING conversion was successful');

TEST_FINISHED();
END_METHOD

METHOD PUBLIC Check_INT_TO_STRING_Max
VAR
	value : INT := DatatypeLimits.INT_MAX_VALUE;
	actual : STRING;
	converted : BOOL;
	equal : BOOL;
END_VAR
TEST('Check_INT_TO_STRING_Max');

// @TEST-RUN
converted := TryConvert_INT_TO_Destination(value, actual);
equal := actual = INT_TO_STRING(value);

// @TEST-ASSERT
AssertTrue(Condition := equal, Message := 'Did not convert INT to STRING correctly');
AssertTrue(Condition := converted, Message := 'Did not report INT to STRING conversion was successful');

TEST_FINISHED();
END_METHOD

METHOD PUBLIC Check_INT_TO_TIME_Min
VAR
	value : INT := DatatypeLimits.MIN_VALUE_OF_INT_WHICH_CAN_BE_HELD_IN_A_TIME;
	actual : TIME;
	converted : BOOL;
	equal : BOOL;
END_VAR
TEST('Check_INT_TO_TIME_Min');

// @TEST-RUN
converted := TryConvert_INT_TO_Destination(value, actual);
equal := actual = INT_TO_TIME(value);

// @TEST-ASSERT
AssertTrue(Condition := equal, Message := 'Did not convert INT to TIME correctly');
AssertTrue(Condition := converted, Message := 'Did not report INT to TIME conversion was successful');

TEST_FINISHED();
END_METHOD

METHOD PUBLIC Check_INT_TO_TIME_TooLow
VAR
	value : INT := DatatypeLimits.INT_MIN_VALUE;
	actual : TIME;
	converted : BOOL;
END_VAR
TEST('Check_INT_TO_TIME_TooLow');

// @TEST-RUN
converted := TryConvert_INT_TO_Destination(value, actual);

// @TEST-ASSERT
AssertFalse(Condition := converted, Message := 'Did not report INT to TIME conversion was prevented');

TEST_FINISHED();
END_METHOD

METHOD PUBLIC Check_INT_TO_TIME_Max
VAR
	value : INT := DatatypeLimits.INT_MAX_VALUE;
	actual : TIME;
	converted : BOOL;
	equal : BOOL;
END_VAR
TEST('Check_INT_TO_TIME_Max');

// @TEST-RUN
converted := TryConvert_INT_TO_Destination(value, actual);
equal := actual = INT_TO_TIME(value);

// @TEST-ASSERT
AssertTrue(Condition := equal, Message := 'Did not convert INT to TIME correctly');
AssertTrue(Condition := converted, Message := 'Did not report INT to TIME conversion was successful');

TEST_FINISHED();
END_METHOD

METHOD PUBLIC Check_INT_TO_TOD_Min
VAR
	value : INT := DatatypeLimits.MIN_VALUE_OF_INT_WHICH_CAN_BE_HELD_IN_A_TOD;
	actual : TOD;
	converted : BOOL;
	equal : BOOL;
END_VAR
TEST('Check_INT_TO_TOD_Min');

// @TEST-RUN
converted := TryConvert_INT_TO_Destination(value, actual);
equal := actual = INT_TO_TOD(value);

// @TEST-ASSERT
AssertTrue(Condition := equal, Message := 'Did not convert INT to TOD correctly');
AssertTrue(Condition := converted, Message := 'Did not report INT to TOD conversion was successful');

TEST_FINISHED();
END_METHOD

METHOD PUBLIC Check_INT_TO_TOD_TooLow
VAR
	value : INT := DatatypeLimits.INT_MIN_VALUE;
	actual : TOD;
	converted : BOOL;
END_VAR
TEST('Check_INT_TO_TOD_TooLow');

// @TEST-RUN
converted := TryConvert_INT_TO_Destination(value, actual);

// @TEST-ASSERT
AssertFalse(Condition := converted, Message := 'Did not report INT to TOD conversion was prevented');

TEST_FINISHED();
END_METHOD

METHOD PUBLIC Check_INT_TO_TOD_Max
VAR
	value : INT := DatatypeLimits.INT_MAX_VALUE;
	actual : TOD;
	converted : BOOL;
	equal : BOOL;
END_VAR
TEST('Check_INT_TO_TOD_Max');

// @TEST-RUN
converted := TryConvert_INT_TO_Destination(value, actual);
equal := actual = INT_TO_TOD(value);

// @TEST-ASSERT
AssertTrue(Condition := equal, Message := 'Did not convert INT to TOD correctly');
AssertTrue(Condition := converted, Message := 'Did not report INT to TOD conversion was successful');

TEST_FINISHED();
END_METHOD

METHOD PUBLIC Check_INT_TO_UDINT_Min
VAR
	value : INT := DatatypeLimits.MIN_VALUE_OF_INT_WHICH_CAN_BE_HELD_IN_A_UDINT;
	actual : UDINT;
	converted : BOOL;
	equal : BOOL;
END_VAR
TEST('Check_INT_TO_UDINT_Min');

// @TEST-RUN
converted := TryConvert_INT_TO_Destination(value, actual);
equal := actual = INT_TO_UDINT(value);

// @TEST-ASSERT
AssertTrue(Condition := equal, Message := 'Did not convert INT to UDINT correctly');
AssertTrue(Condition := converted, Message := 'Did not report INT to UDINT conversion was successful');

TEST_FINISHED();
END_METHOD

METHOD PUBLIC Check_INT_TO_UDINT_TooLow
VAR
	value : INT := DatatypeLimits.INT_MIN_VALUE;
	actual : UDINT;
	converted : BOOL;
END_VAR
TEST('Check_INT_TO_UDINT_TooLow');

// @TEST-RUN
converted := TryConvert_INT_TO_Destination(value, actual);

// @TEST-ASSERT
AssertFalse(Condition := converted, Message := 'Did not report INT to UDINT conversion was prevented');

TEST_FINISHED();
END_METHOD

METHOD PUBLIC Check_INT_TO_UDINT_Max
VAR
	value : INT := DatatypeLimits.INT_MAX_VALUE;
	actual : UDINT;
	converted : BOOL;
	equal : BOOL;
END_VAR
TEST('Check_INT_TO_UDINT_Max');

// @TEST-RUN
converted := TryConvert_INT_TO_Destination(value, actual);
equal := actual = INT_TO_UDINT(value);

// @TEST-ASSERT
AssertTrue(Condition := equal, Message := 'Did not convert INT to UDINT correctly');
AssertTrue(Condition := converted, Message := 'Did not report INT to UDINT conversion was successful');

TEST_FINISHED();
END_METHOD

METHOD PUBLIC Check_INT_TO_UINT_Min
VAR
	value : INT := DatatypeLimits.MIN_VALUE_OF_INT_WHICH_CAN_BE_HELD_IN_A_UINT;
	actual : UINT;
	converted : BOOL;
	equal : BOOL;
END_VAR
TEST('Check_INT_TO_UINT_Min');

// @TEST-RUN
converted := TryConvert_INT_TO_Destination(value, actual);
equal := actual = INT_TO_UINT(value);

// @TEST-ASSERT
AssertTrue(Condition := equal, Message := 'Did not convert INT to UINT correctly');
AssertTrue(Condition := converted, Message := 'Did not report INT to UINT conversion was successful');

TEST_FINISHED();
END_METHOD

METHOD PUBLIC Check_INT_TO_UINT_TooLow
VAR
	value : INT := DatatypeLimits.INT_MIN_VALUE;
	actual : UINT;
	converted : BOOL;
END_VAR
TEST('Check_INT_TO_UINT_TooLow');

// @TEST-RUN
converted := TryConvert_INT_TO_Destination(value, actual);

// @TEST-ASSERT
AssertFalse(Condition := converted, Message := 'Did not report INT to UINT conversion was prevented');

TEST_FINISHED();
END_METHOD

METHOD PUBLIC Check_INT_TO_UINT_Max
VAR
	value : INT := DatatypeLimits.INT_MAX_VALUE;
	actual : UINT;
	converted : BOOL;
	equal : BOOL;
END_VAR
TEST('Check_INT_TO_UINT_Max');

// @TEST-RUN
converted := TryConvert_INT_TO_Destination(value, actual);
equal := actual = INT_TO_UINT(value);

// @TEST-ASSERT
AssertTrue(Condition := equal, Message := 'Did not convert INT to UINT correctly');
AssertTrue(Condition := converted, Message := 'Did not report INT to UINT conversion was successful');

TEST_FINISHED();
END_METHOD

METHOD PUBLIC Check_INT_TO_ULINT_Min
VAR
	value : INT := DatatypeLimits.MIN_VALUE_OF_INT_WHICH_CAN_BE_HELD_IN_A_ULINT;
	actual : ULINT;
	converted : BOOL;
	equal : BOOL;
END_VAR
TEST('Check_INT_TO_ULINT_Min');

// @TEST-RUN
converted := TryConvert_INT_TO_Destination(value, actual);
equal := actual = INT_TO_ULINT(value);

// @TEST-ASSERT
AssertTrue(Condition := equal, Message := 'Did not convert INT to ULINT correctly');
AssertTrue(Condition := converted, Message := 'Did not report INT to ULINT conversion was successful');

TEST_FINISHED();
END_METHOD

METHOD PUBLIC Check_INT_TO_ULINT_TooLow
VAR
	value : INT := DatatypeLimits.INT_MIN_VALUE;
	actual : ULINT;
	converted : BOOL;
END_VAR
TEST('Check_INT_TO_ULINT_TooLow');

// @TEST-RUN
converted := TryConvert_INT_TO_Destination(value, actual);

// @TEST-ASSERT
AssertFalse(Condition := converted, Message := 'Did not report INT to ULINT conversion was prevented');

TEST_FINISHED();
END_METHOD

METHOD PUBLIC Check_INT_TO_ULINT_Max
VAR
	value : INT := DatatypeLimits.INT_MAX_VALUE;
	actual : ULINT;
	converted : BOOL;
	equal : BOOL;
END_VAR
TEST('Check_INT_TO_ULINT_Max');

// @TEST-RUN
converted := TryConvert_INT_TO_Destination(value, actual);
equal := actual = INT_TO_ULINT(value);

// @TEST-ASSERT
AssertTrue(Condition := equal, Message := 'Did not convert INT to ULINT correctly');
AssertTrue(Condition := converted, Message := 'Did not report INT to ULINT conversion was successful');

TEST_FINISHED();
END_METHOD

METHOD PUBLIC Check_INT_TO_USINT_Min
VAR
	value : INT := DatatypeLimits.MIN_VALUE_OF_INT_WHICH_CAN_BE_HELD_IN_A_USINT;
	actual : USINT;
	converted : BOOL;
	equal : BOOL;
END_VAR
TEST('Check_INT_TO_USINT_Min');

// @TEST-RUN
converted := TryConvert_INT_TO_Destination(value, actual);
equal := actual = INT_TO_USINT(value);

// @TEST-ASSERT
AssertTrue(Condition := equal, Message := 'Did not convert INT to USINT correctly');
AssertTrue(Condition := converted, Message := 'Did not report INT to USINT conversion was successful');

TEST_FINISHED();
END_METHOD

METHOD PUBLIC Check_INT_TO_USINT_TooHigh
VAR
	value : INT := DatatypeLimits.INT_MAX_VALUE;
	actual : USINT;
	converted : BOOL;
END_VAR
TEST('Check_INT_TO_USINT_TooHigh');

// @TEST-RUN
converted := TryConvert_INT_TO_Destination(value, actual);

// @TEST-ASSERT
AssertFalse(Condition := converted, Message := 'Did not report INT to USINT conversion was prevented');

TEST_FINISHED();
END_METHOD

METHOD PUBLIC Check_INT_TO_USINT_TooLow
VAR
	value : INT := DatatypeLimits.INT_MIN_VALUE;
	actual : USINT;
	converted : BOOL;
END_VAR
TEST('Check_INT_TO_USINT_TooLow');

// @TEST-RUN
converted := TryConvert_INT_TO_Destination(value, actual);

// @TEST-ASSERT
AssertFalse(Condition := converted, Message := 'Did not report INT to USINT conversion was prevented');

TEST_FINISHED();
END_METHOD

METHOD PUBLIC Check_INT_TO_USINT_Max
VAR
	value : INT := DatatypeLimits.MAX_VALUE_OF_INT_WHICH_CAN_BE_HELD_IN_A_USINT;
	actual : USINT;
	converted : BOOL;
	equal : BOOL;
END_VAR
TEST('Check_INT_TO_USINT_Max');

// @TEST-RUN
converted := TryConvert_INT_TO_Destination(value, actual);
equal := actual = INT_TO_USINT(value);

// @TEST-ASSERT
AssertTrue(Condition := equal, Message := 'Did not convert INT to USINT correctly');
AssertTrue(Condition := converted, Message := 'Did not report INT to USINT conversion was successful');

TEST_FINISHED();
END_METHOD

METHOD PUBLIC Check_INT_TO_WORD_Min
VAR
	value : INT := DatatypeLimits.MIN_VALUE_OF_INT_WHICH_CAN_BE_HELD_IN_A_WORD;
	actual : WORD;
	converted : BOOL;
	equal : BOOL;
END_VAR
TEST('Check_INT_TO_WORD_Min');

// @TEST-RUN
converted := TryConvert_INT_TO_Destination(value, actual);
equal := actual = INT_TO_WORD(value);

// @TEST-ASSERT
AssertTrue(Condition := equal, Message := 'Did not convert INT to WORD correctly');
AssertTrue(Condition := converted, Message := 'Did not report INT to WORD conversion was successful');

TEST_FINISHED();
END_METHOD

METHOD PUBLIC Check_INT_TO_WORD_TooLow
VAR
	value : INT := DatatypeLimits.INT_MIN_VALUE;
	actual : WORD;
	converted : BOOL;
END_VAR
TEST('Check_INT_TO_WORD_TooLow');

// @TEST-RUN
converted := TryConvert_INT_TO_Destination(value, actual);

// @TEST-ASSERT
AssertFalse(Condition := converted, Message := 'Did not report INT to WORD conversion was prevented');

TEST_FINISHED();
END_METHOD

METHOD PUBLIC Check_INT_TO_WORD_Max
VAR
	value : INT := DatatypeLimits.INT_MAX_VALUE;
	actual : WORD;
	converted : BOOL;
	equal : BOOL;
END_VAR
TEST('Check_INT_TO_WORD_Max');

// @TEST-RUN
converted := TryConvert_INT_TO_Destination(value, actual);
equal := actual = INT_TO_WORD(value);

// @TEST-ASSERT
AssertTrue(Condition := equal, Message := 'Did not convert INT to WORD correctly');
AssertTrue(Condition := converted, Message := 'Did not report INT to WORD conversion was successful');

TEST_FINISHED();
END_METHOD

END_FUNCTION_BLOCK

// ---- Tests/DINT_TO_TestSuite.TcPOU
FUNCTION_BLOCK PUBLIC DINT_TO_TestSuite EXTENDS TcUnit.FB_TestSuite
VAR
END_VAR

Check_DINT_TO_BOOL_Max();
Check_DINT_TO_BOOL_Min();
Check_DINT_TO_BYTE_Max();
Check_DINT_TO_BYTE_Min();
Check_DINT_TO_BYTE_TooHigh();
Check_DINT_TO_BYTE_TooLow();
Check_DINT_TO_WORD_Max();
Check_DINT_TO_WORD_Min();
Check_DINT_TO_WORD_TooHigh();
Check_DINT_TO_WORD_TooLow();
Check_DINT_TO_DWORD_Max();
Check_DINT_TO_DWORD_Min();
Check_DINT_TO_DWORD_TooLow();
Check_DINT_TO_LWORD_Max();
Check_DINT_TO_LWORD_Min();
Check_DINT_TO_LWORD_TooLow();
Check_DINT_TO_SINT_Max();
Check_DINT_TO_SINT_Min();
Check_DINT_TO_SINT_TooHigh();
Check_DINT_TO_SINT_TooLow();
Check_DINT_TO_INT_Max();
Check_DINT_TO_INT_Min();
Check_DINT_TO_INT_TooHigh();
Check_DINT_TO_INT_TooLow();
Check_DINT_TO_DINT_Max();
Check_DINT_TO_DINT_Min();
Check_DINT_TO_LINT_Max();
Check_DINT_TO_LINT_Min();
Check_DINT_TO_USINT_Max();
Check_DINT_TO_USINT_Min();
Check_DINT_TO_USINT_TooHigh();
Check_DINT_TO_USINT_TooLow();
Check_DINT_TO_UINT_Max();
Check_DINT_TO_UINT_Min();
Check_DINT_TO_UINT_TooHigh();
Check_DINT_TO_UINT_TooLow();
Check_DINT_TO_UDINT_Max();
Check_DINT_TO_UDINT_Min();
Check_DINT_TO_UDINT_TooLow();
Check_DINT_TO_ULINT_Max();
Check_DINT_TO_ULINT_Min();
Check_DINT_TO_ULINT_TooLow();
Check_DINT_TO_REAL_Max();
Check_DINT_TO_REAL_Min();
Check_DINT_TO_LREAL_Max();
Check_DINT_TO_LREAL_Min();
Check_DINT_TO_TIME_Max();
Check_DINT_TO_TIME_Min();
Check_DINT_TO_TIME_TooLow();
Check_DINT_TO_TOD_Max();
Check_DINT_TO_TOD_Min();
Check_DINT_TO_TOD_TooHigh();
Check_DINT_TO_TOD_TooLow();
Check_DINT_TO_DATE_Max();
Check_DINT_TO_DATE_Min();
Check_DINT_TO_DATE_TooLow();
Check_DINT_TO_DT_Max();
Check_DINT_TO_DT_Min();
Check_DINT_TO_DT_TooLow();
Check_DINT_TO_STRING_Max();
Check_DINT_TO_STRING_Min();

METHOD PUBLIC Check_DINT_TO_BOOL_Min
VAR
	value : DINT := DatatypeLimits.DINT_MIN_VALUE;
	actual : BOOL;
	converted : BOOL;
	equal : BOOL;
END_VAR
TEST('Check_DINT_TO_BOOL_Min');

// @TEST-RUN
converted := TryConvert_DINT_TO_Destination(value, actual);
equal := actual = DINT_TO_BOOL(value);

// @TEST-ASSERT
AssertTrue(Condition := equal, Message := 'Did not convert DINT to BOOL correctly');
AssertTrue(Condition := converted, Message := 'Did not report DINT to BOOL conversion was successful');

TEST_FINISHED();
END_METHOD

METHOD PUBLIC Check_DINT_TO_BOOL_Max
VAR
	value : DINT := DatatypeLimits.DINT_MAX_VALUE;
	actual : BOOL;
	converted : BOOL;
	equal : BOOL;
END_VAR
TEST('Check_DINT_TO_BOOL_Max');

// @TEST-RUN
converted := TryConvert_DINT_TO_Destination(value, actual);
equal := actual = DINT_TO_BOOL(value);

// @TEST-ASSERT
AssertTrue(Condition := equal, Message := 'Did not convert DINT to BOOL correctly');
AssertTrue(Condition := converted, Message := 'Did not report DINT to BOOL conversion was successful');

TEST_FINISHED();
END_METHOD

METHOD PUBLIC Check_DINT_TO_BYTE_Min
VAR
	value : DINT := DatatypeLimits.MIN_VALUE_OF_DINT_WHICH_CAN_BE_HELD_IN_A_BYTE;
	actual : BYTE;
	converted : BOOL;
	equal : BOOL;
END_VAR
TEST('Check_DINT_TO_BYTE_Min');

// @TEST-RUN
converted := TryConvert_DINT_TO_Destination(value, actual);
equal := actual = DINT_TO_BYTE(value);

// @TEST-ASSERT
AssertTrue(Condition := equal, Message := 'Did not convert DINT to BYTE correctly');
AssertTrue(Condition := converted, Message := 'Did not report DINT to BYTE conversion was successful');

TEST_FINISHED();
END_METHOD

METHOD PUBLIC Check_DINT_TO_BYTE_TooHigh
VAR
	value : DINT := DatatypeLimits.DINT_MAX_VALUE;
	actual : BYTE;
	converted : BOOL;
END_VAR
TEST('Check_DINT_TO_BYTE_TooHigh');

// @TEST-RUN
converted := TryConvert_DINT_TO_Destination(value, actual);

// @TEST-ASSERT
AssertFalse(Condition := converted, Message := 'Did not report DINT to BYTE conversion was prevented');

TEST_FINISHED();
END_METHOD

METHOD PUBLIC Check_DINT_TO_BYTE_TooLow
VAR
	value : DINT := DatatypeLimits.DINT_MIN_VALUE;
	actual : BYTE;
	converted : BOOL;
END_VAR
TEST('Check_DINT_TO_BYTE_TooLow');

// @TEST-RUN
converted := TryConvert_DINT_TO_Destination(value, actual);

// @TEST-ASSERT
AssertFalse(Condition := converted, Message := 'Did not report DINT to BYTE conversion was prevented');

TEST_FINISHED();
END_METHOD

METHOD PUBLIC Check_DINT_TO_BYTE_Max
VAR
	value : DINT := DatatypeLimits.MAX_VALUE_OF_DINT_WHICH_CAN_BE_HELD_IN_A_BYTE;
	actual : BYTE;
	converted : BOOL;
	equal : BOOL;
END_VAR
TEST('Check_DINT_TO_BYTE_Max');

// @TEST-RUN
converted := TryConvert_DINT_TO_Destination(value, actual);
equal := actual = DINT_TO_BYTE(value);

// @TEST-ASSERT
AssertTrue(Condition := equal, Message := 'Did not convert DINT to BYTE correctly');
AssertTrue(Condition := converted, Message := 'Did not report DINT to BYTE conversion was successful');

TEST_FINISHED();
END_METHOD

METHOD PUBLIC Check_DINT_TO_DATE_Min
VAR
	value : DINT := DatatypeLimits.MIN_VALUE_OF_DINT_WHICH_CAN_BE_HELD_IN_A_DATE;
	actual : DATE;
	converted : BOOL;
	equal : BOOL;
END_VAR
TEST('Check_DINT_TO_DATE_Min');

// @TEST-RUN
converted := TryConvert_DINT_TO_Destination(value, actual);
equal := actual = DINT_TO_DATE(value);

// @TEST-ASSERT
AssertTrue(Condition := equal, Message := 'Did not convert DINT to DATE correctly');
AssertTrue(Condition := converted, Message := 'Did not report DINT to DATE conversion was successful');

TEST_FINISHED();
END_METHOD

METHOD PUBLIC Check_DINT_TO_DATE_TooLow
VAR
	value : DINT := DatatypeLimits.DINT_MIN_VALUE;
	actual : DATE;
	converted : BOOL;
END_VAR
TEST('Check_DINT_TO_DATE_TooLow');

// @TEST-RUN
converted := TryConvert_DINT_TO_Destination(value, actual);

// @TEST-ASSERT
AssertFalse(Condition := converted, Message := 'Did not report DINT to DATE conversion was prevented');

TEST_FINISHED();
END_METHOD

METHOD PUBLIC Check_DINT_TO_DATE_Max
VAR
	value : DINT := DatatypeLimits.DINT_MAX_VALUE;
	actual : DATE;
	converted : BOOL;
	equal : BOOL;
END_VAR
TEST('Check_DINT_TO_DATE_Max');

// @TEST-RUN
converted := TryConvert_DINT_TO_Destination(value, actual);
equal := actual = DINT_TO_DATE(value);

// @TEST-ASSERT
AssertTrue(Condition := equal, Message := 'Did not convert DINT to DATE correctly');
AssertTrue(Condition := converted, Message := 'Did not report DINT to DATE conversion was successful');

TEST_FINISHED();
END_METHOD

METHOD PUBLIC Check_DINT_TO_DINT_Min
VAR
	value : DINT := DatatypeLimits.DINT_MIN_VALUE;
	actual : DINT;
	converted : BOOL;
	equal : BOOL;
END_VAR
TEST('Check_DINT_TO_DINT_Min');

// @TEST-RUN
converted := TryConvert_DINT_TO_Destination(value, actual);
equal := actual = value;

// @TEST-ASSERT
AssertTrue(Condition := equal, Message := 'Did not convert DINT to DINT correctly');
AssertTrue(Condition := converted, Message := 'Did not report DINT to DINT conversion was successful');

TEST_FINISHED();
END_METHOD

METHOD PUBLIC Check_DINT_TO_DINT_Max
VAR
	value : DINT := DatatypeLimits.DINT_MAX_VALUE;
	actual : DINT;
	converted : BOOL;
	equal : BOOL;
END_VAR
TEST('Check_DINT_TO_DINT_Max');

// @TEST-RUN
converted := TryConvert_DINT_TO_Destination(value, actual);
equal := actual = value;

// @TEST-ASSERT
AssertTrue(Condition := equal, Message := 'Did not convert DINT to DINT correctly');
AssertTrue(Condition := converted, Message := 'Did not report DINT to DINT conversion was successful');

TEST_FINISHED();
END_METHOD

METHOD PUBLIC Check_DINT_TO_DT_Min
VAR
	value : DINT := DatatypeLimits.MIN_VALUE_OF_DINT_WHICH_CAN_BE_HELD_IN_A_DT;
	actual : DT;
	converted : BOOL;
	equal : BOOL;
END_VAR
TEST('Check_DINT_TO_DT_Min');

// @TEST-RUN
converted := TryConvert_DINT_TO_Destination(value, actual);
equal := actual = DINT_TO_DT(value);

// @TEST-ASSERT
AssertTrue(Condition := equal, Message := 'Did not convert DINT to DT correctly');
AssertTrue(Condition := converted, Message := 'Did not report DINT to DT conversion was successful');

TEST_FINISHED();
END_METHOD

METHOD PUBLIC Check_DINT_TO_DT_TooLow
VAR
	value : DINT := DatatypeLimits.DINT_MIN_VALUE;
	actual : DT;
	converted : BOOL;
END_VAR
TEST('Check_DINT_TO_DT_TooLow');

// @TEST-RUN
converted := TryConvert_DINT_TO_Destination(value, actual);

// @TEST-ASSERT
AssertFalse(Condition := converted, Message := 'Did not report DINT to DT conversion was prevented');

TEST_FINISHED();
END_METHOD

METHOD PUBLIC Check_DINT_TO_DT_Max
VAR
	value : DINT := DatatypeLimits.DINT_MAX_VALUE;
	actual : DT;
	converted : BOOL;
	equal : BOOL;
END_VAR
TEST('Check_DINT_TO_DT_Max');

// @TEST-RUN
converted := TryConvert_DINT_TO_Destination(value, actual);
equal := actual = DINT_TO_DT(value);

// @TEST-ASSERT
AssertTrue(Condition := equal, Message := 'Did not convert DINT to DT correctly');
AssertTrue(Condition := converted, Message := 'Did not report DINT to DT conversion was successful');

TEST_FINISHED();
END_METHOD

METHOD PUBLIC Check_DINT_TO_DWORD_Min
VAR
	value : DINT := DatatypeLimits.MIN_VALUE_OF_DINT_WHICH_CAN_BE_HELD_IN_A_DWORD;
	actual : DWORD;
	converted : BOOL;
	equal : BOOL;
END_VAR
TEST('Check_DINT_TO_DWORD_Min');

// @TEST-RUN
converted := TryConvert_DINT_TO_Destination(value, actual);
equal := actual = DINT_TO_DWORD(value);

// @TEST-ASSERT
AssertTrue(Condition := equal, Message := 'Did not convert DINT to DWORD correctly');
AssertTrue(Condition := converted, Message := 'Did not report DINT to DWORD conversion was successful');

TEST_FINISHED();
END_METHOD

METHOD PUBLIC Check_DINT_TO_DWORD_TooLow
VAR
	value : DINT := DatatypeLimits.DINT_MIN_VALUE;
	actual : DWORD;
	converted : BOOL;
END_VAR
TEST('Check_DINT_TO_DWORD_TooLow');

// @TEST-RUN
converted := TryConvert_DINT_TO_Destination(value, actual);

// @TEST-ASSERT
AssertFalse(Condition := converted, Message := 'Did not report DINT to DWORD conversion was prevented');

TEST_FINISHED();
END_METHOD

METHOD PUBLIC Check_DINT_TO_DWORD_Max
VAR
	value : DINT := DatatypeLimits.DINT_MAX_VALUE;
	actual : DWORD;
	converted : BOOL;
	equal : BOOL;
END_VAR
TEST('Check_DINT_TO_DWORD_Max');

// @TEST-RUN
converted := TryConvert_DINT_TO_Destination(value, actual);
equal := actual = DINT_TO_DWORD(value);

// @TEST-ASSERT
AssertTrue(Condition := equal, Message := 'Did not convert DINT to DWORD correctly');
AssertTrue(Condition := converted, Message := 'Did not report DINT to DWORD conversion was successful');

TEST_FINISHED();
END_METHOD

METHOD PUBLIC Check_DINT_TO_INT_Min
VAR
	value : DINT := DatatypeLimits.MIN_VALUE_OF_DINT_WHICH_CAN_BE_HELD_IN_A_INT;
	actual : INT;
	converted : BOOL;
	equal : BOOL;
END_VAR
TEST('Check_DINT_TO_INT_Min');

// @TEST-RUN
converted := TryConvert_DINT_TO_Destination(value, actual);
equal := actual = DINT_TO_INT(value);

// @TEST-ASSERT
AssertTrue(Condition := equal, Message := 'Did not convert DINT to INT correctly');
AssertTrue(Condition := converted, Message := 'Did not report DINT to INT conversion was successful');

TEST_FINISHED();
END_METHOD

METHOD PUBLIC Check_DINT_TO_INT_TooHigh
VAR
	value : DINT := DatatypeLimits.DINT_MAX_VALUE;
	actual : INT;
	converted : BOOL;
END_VAR
TEST('Check_DINT_TO_INT_TooHigh');

// @TEST-RUN
converted := TryConvert_DINT_TO_Destination(value, actual);

// @TEST-ASSERT
AssertFalse(Condition := converted, Message := 'Did not report DINT to INT conversion was prevented');

TEST_FINISHED();
END_METHOD

METHOD PUBLIC Check_DINT_TO_INT_TooLow
VAR
	value : DINT := DatatypeLimits.DINT_MIN_VALUE;
	actual : INT;
	converted : BOOL;
END_VAR
TEST('Check_DINT_TO_INT_TooLow');

// @TEST-RUN
converted := TryConvert_DINT_TO_Destination(value, actual);

// @TEST-ASSERT
AssertFalse(Condition := converted, Message := 'Did not report DINT to INT conversion was prevented');

TEST_FINISHED();
END_METHOD

METHOD PUBLIC Check_DINT_TO_INT_Max
VAR
	value : DINT := DatatypeLimits.MAX_VALUE_OF_DINT_WHICH_CAN_BE_HELD_IN_A_INT;
	actual : INT;
	converted : BOOL;
	equal : BOOL;
END_VAR
TEST('Check_DINT_TO_INT_Max');

// @TEST-RUN
converted := TryConvert_DINT_TO_Destination(value, actual);
equal := actual = DINT_TO_INT(value);

// @TEST-ASSERT
AssertTrue(Condition := equal, Message := 'Did not convert DINT to INT correctly');
AssertTrue(Condition := converted, Message := 'Did not report DINT to INT conversion was successful');

TEST_FINISHED();
END_METHOD

METHOD PUBLIC Check_DINT_TO_LINT_Min
VAR
	value : DINT := DatatypeLimits.DINT_MIN_VALUE;
	actual : LINT;
	converted : BOOL;
	equal : BOOL;
END_VAR
TEST('Check_DINT_TO_LINT_Min');

// @TEST-RUN
converted := TryConvert_DINT_TO_Destination(value, actual);
equal := actual = DINT_TO_LINT(value);

// @TEST-ASSERT
AssertTrue(Condition := equal, Message := 'Did not convert DINT to LINT correctly');
AssertTrue(Condition := converted, Message := 'Did not report DINT to LINT conversion was successful');

TEST_FINISHED();
END_METHOD

METHOD PUBLIC Check_DINT_TO_LINT_Max
VAR
	value : DINT := DatatypeLimits.DINT_MAX_VALUE;
	actual : LINT;
	converted : BOOL;
	equal : BOOL;
END_VAR
TEST('Check_DINT_TO_LINT_Max');

// @TEST-RUN
converted := TryConvert_DINT_TO_Destination(value, actual);
equal := actual = DINT_TO_LINT(value);

// @TEST-ASSERT
AssertTrue(Condition := equal, Message := 'Did not convert DINT to LINT correctly');
AssertTrue(Condition := converted, Message := 'Did not report DINT to LINT conversion was successful');

TEST_FINISHED();
END_METHOD

METHOD PUBLIC Check_DINT_TO_LREAL_Min
VAR
	value : DINT := DatatypeLimits.DINT_MIN_VALUE;
	actual : LREAL;
	converted : BOOL;
	equal : BOOL;
END_VAR
TEST('Check_DINT_TO_LREAL_Min');

// @TEST-RUN
converted := TryConvert_DINT_TO_Destination(value, actual);
equal := actual = DINT_TO_LREAL(value);

// @TEST-ASSERT
AssertTrue(Condition := equal, Message := 'Did not convert DINT to LREAL correctly');
AssertTrue(Condition := converted, Message := 'Did not report DINT to LREAL conversion was successful');

TEST_FINISHED();
END_METHOD

METHOD PUBLIC Check_DINT_TO_LREAL_Max
VAR
	value : DINT := DatatypeLimits.DINT_MAX_VALUE;
	actual : LREAL;
	converted : BOOL;
	equal : BOOL;
END_VAR
TEST('Check_DINT_TO_LREAL_Max');

// @TEST-RUN
converted := TryConvert_DINT_TO_Destination(value, actual);
equal := actual = DINT_TO_LREAL(value);

// @TEST-ASSERT
AssertTrue(Condition := equal, Message := 'Did not convert DINT to LREAL correctly');
AssertTrue(Condition := converted, Message := 'Did not report DINT to LREAL conversion was successful');

TEST_FINISHED();
END_METHOD

METHOD PUBLIC Check_DINT_TO_LWORD_Min
VAR
	value : DINT := DatatypeLimits.MIN_VALUE_OF_DINT_WHICH_CAN_BE_HELD_IN_A_LWORD;
	actual : LWORD;
	converted : BOOL;
	equal : BOOL;
END_VAR
TEST('Check_DINT_TO_LWORD_Min');

// @TEST-RUN
converted := TryConvert_DINT_TO_Destination(value, actual);
equal := actual = DINT_TO_LWORD(value);

// @TEST-ASSERT
AssertTrue(Condition := equal, Message := 'Did not convert DINT to LWORD correctly');
AssertTrue(Condition := converted, Message := 'Did not report DINT to LWORD conversion was successful');

TEST_FINISHED();
END_METHOD

METHOD PUBLIC Check_DINT_TO_LWORD_TooLow
VAR
	value : DINT := DatatypeLimits.DINT_MIN_VALUE;
	actual : LWORD;
	converted : BOOL;
END_VAR
TEST('Check_DINT_TO_LWORD_TooLow');

// @TEST-RUN
converted := TryConvert_DINT_TO_Destination(value, actual);

// @TEST-ASSERT
AssertFalse(Condition := converted, Message := 'Did not report DINT to LWORD conversion was prevented');

TEST_FINISHED();
END_METHOD

METHOD PUBLIC Check_DINT_TO_LWORD_Max
VAR
	value : DINT := DatatypeLimits.DINT_MAX_VALUE;
	actual : LWORD;
	converted : BOOL;
	equal : BOOL;
END_VAR
TEST('Check_DINT_TO_LWORD_Max');

// @TEST-RUN
converted := TryConvert_DINT_TO_Destination(value, actual);
equal := actual = DINT_TO_LWORD(value);

// @TEST-ASSERT
AssertTrue(Condition := equal, Message := 'Did not convert DINT to LWORD correctly');
AssertTrue(Condition := converted, Message := 'Did not report DINT to LWORD conversion was successful');

TEST_FINISHED();
END_METHOD

METHOD PUBLIC Check_DINT_TO_REAL_Min
VAR
	value : DINT := DatatypeLimits.DINT_MIN_VALUE;
	actual : REAL;
	converted : BOOL;
	equal : BOOL;
END_VAR
TEST('Check_DINT_TO_REAL_Min');

// @TEST-RUN
converted := TryConvert_DINT_TO_Destination(value, actual);
equal := actual = DINT_TO_REAL(value);

